// SIMATIC STEP 7 (V5.x) project newgenpns
// station: Hardware
// station: SIMATIC 300(1)
// station: P_ADR_BUS
// station: P_ADR_BUS
// station: Configuration
// program: S7 Program(1)

SYMBOL_TABLE
"PressDB"	DB 3	DB 3
"FCs"	DB 4	DB 4
"NOMINAL"	DB 71	DB 71
"EtoDBfunc"	DB 97	DB 97
"AtoDBfunc"	DB 98	DB 98
"AlarmState"	DB 99	DB 99
"Alarms"	DB 101	DB 101
"mada"	DB 102	DB 102
"Events"	DB 111	DB 111
"DB_ROTATION"	DB 200	DB 200
"PROCESS_DATA"	DB 300	DB 300
"kagiri"	DB 302	DB 302
"DB_PUMPOFF"	DB 303	DB 303
"MM430_NS1"	DB 500	DB 500
"Scale"	FC 3	FC 3
"FaultCheck"	FC 5	FC 5
"DT to DATE"	FC 6	FC 6	// DT to DATE
"DT to DAY"	FC 7	FC 7	// DT to DAY
"DT to TOD"	FC 8	FC 8	// DT to TOD
"GE_DT"	FC 12	FC 12	// Greater or Equal DT
"EventsCheck"	FC 55	FC 55
"DATE and TOD to DT"	FC 62	FC 62	// Date and TOD to DT
"rawConvert"	FC 100	FC 100
"aisConvert"	FC 102	FC 102
"maCalibration"	FC 103	FC 103
"FAULT_CHECK"	FC 105	FC 105
"AlarmToDB"	FC 106	FC 106
"Copyd"	FC 107	FC 107
"ToPanel"	FC 108	FC 108
"EventToDB"	FC 116	FC 116
"Copyb"	FC 117	FC 117
"EToPanel"	FC 118	FC 118
"date&time"	FC 121	FC 121
"ROTATION"	FC 200	FC 200
"PNS_CORE"	FC 300	FC 300
"PUMPS_TOGGLE"	FC 301	FC 301
"FICTION_PRIORITY"	FC 302	FC 302
"MICROMASTER_4XX"	FC 500	FC 500
"Fire"	I 1.0	BOOL
"Security"	I 1.1	BOOL
"Overflow"	I 1.2	BOOL
"Phase"	I 1.3	BOOL
"Input1AVR"	I 2.0	BOOL
"Input2AVR"	I 2.1	BOOL
"Mushroom"	I 2.2	BOOL
"Dryhot"	I 2.3	BOOL
"DI_p1_confirm"	I 3.0	BOOL
"DI_p2_confirm"	I 3.1	BOOL
"DI_p3_confirm"	I 3.2	BOOL
"DI_p4_confirm"	I 3.3	BOOL
"DI_p5_confirm"	I 4.0	BOOL
"DI_p6_confirm"	I 4.1	BOOL
"DI_p1_auto"	I 4.2	BOOL
"DI_p2_auto"	I 4.3	BOOL
"DI_p3_auto"	I 10.0	BOOL
"DI_p4_auto"	I 10.1	BOOL
"pmp1turnOn"	M 13.0	BOOL
"pmp3turnOn"	M 13.1	BOOL
"pmp2turnOn"	M 13.2	BOOL
"RESERVE_BIT"	M 13.3	BOOL
"pmp4turnOn"	M 13.4	BOOL
"SFM0"	M 15.0	BOOL
"SFM1"	M 15.1	BOOL
"SFM2"	M 15.2	BOOL
"SFM3"	M 15.3	BOOL
"EM1"	M 50.0	BOOL
"EM2"	M 50.1	BOOL
"EM3"	M 50.2	BOOL
"EM4"	M 50.3	BOOL
"EM5"	M 50.4	BOOL
"EM6"	M 50.5	BOOL
"EM7"	M 50.6	BOOL
"EM8"	M 50.7	BOOL
"EM9"	M 51.0	BOOL
"EM10"	M 51.1	BOOL
"EM11"	M 51.2	BOOL
"EM12"	M 51.3	BOOL
"starterFPbegin"	M 60.0	BOOL
"starterFPend"	M 60.1	BOOL
"IN_p1_start"	M 70.0	BOOL
"IN_p2_start"	M 70.1	BOOL
"IN_p3_start"	M 70.2	BOOL
"miAuto1"	M 70.3	BOOL
"miAuto2"	M 70.4	BOOL
"miAuto3"	M 70.5	BOOL
"miAuto4"	M 70.6	BOOL
"fcM11"	M 70.7	BOOL
"fcM12"	M 71.0	BOOL
"fcM13"	M 71.1	BOOL
"fcM14"	M 71.2	BOOL
"fcM15"	M 71.3	BOOL
"fcM16"	M 71.4	BOOL
"fcM17"	M 71.5	BOOL
"guuzenFP1"	M 71.6	BOOL
"guuzenFP2"	M 71.7	BOOL
"guuzenFP3"	M 72.0	BOOL
"guuzenFP4"	M 72.1	BOOL
"fcM18"	M 72.2	BOOL
"fcM19"	M 72.3	BOOL
"fcM20"	M 72.4	BOOL
"fcM21"	M 72.5	BOOL
"fcM22"	M 72.6	BOOL
"fcM1"	M 72.7	BOOL
"fcM2"	M 73.0	BOOL
"fcM3"	M 73.1	BOOL
"fcM4"	M 73.2	BOOL
"fcM5"	M 73.3	BOOL
"fcM6"	M 73.4	BOOL
"fcM7"	M 73.5	BOOL
"fcM8"	M 73.6	BOOL
"fcM9"	M 73.7	BOOL
"fcM10"	M 74.0	BOOL
"rotFPbegin"	M 80.0	BOOL
"rotSwiMode"	M 122.0	BOOL
"timeHasCome"	M 122.1	BOOL
"rotation200"	M 122.2	BOOL
"pInput"	PIW 368	WORD
"pOutput"	PIW 370	WORD
"DO_alarm"	Q 4.0	BOOL
"DO_dry"	Q 4.1	BOOL
"DO_p1_turnOn"	Q 6.0	BOOL
"DO_p2_turnOn"	Q 6.1	BOOL
"DO_p3_turnOn"	Q 7.0	BOOL
"DO_p4_turnOn"	Q 7.1	BOOL
"SET_CLK"	SFC 0	SFC 0	// Set System Clock
"READ_CLK"	SFC 1	SFC 1	// Read System Clock
"DPRD_DAT"	SFC 14	SFC 14	// Read Consistent Data of a Standard DP Slave
"DPWR_DAT"	SFC 15	SFC 15	// Write Consistent Data to a Standard DP Slave
"main_started"	T 1	TIMER
"reserve_started"	T 2	TIMER
"lowPressTimer"	T 3	TIMER
"delayStartMain"	T 4	TIMER
"delayStartRes"	T 5	TIMER
"delayStartSRes"	T 6	TIMER
"reserve_stopped"	T 7	TIMER
"second_res_stopped"	T 8	TIMER
"highPressTimer"	T 9	TIMER
"silentRot"	T 10	TIMER
"fcTimer1"	T 13	TIMER
"fcTimer2"	T 14	TIMER
"fcTimer3"	T 15	TIMER
"fcTimer4"	T 16	TIMER
"p2_guuzenTimer"	T 17	TIMER
"p3_guuzenTimer"	T 18	TIMER
"fcTimer9"	T 19	TIMER
"fcTimer10"	T 20	TIMER
"fcTimer5"	T 37	TIMER
"fcTimer6"	T 38	TIMER
"fcTimer7"	T 39	TIMER
"fcTimer8"	T 40	TIMER
"mainFC1_20Hz"	T 41	TIMER
"mainFC2_20Hz"	T 42	TIMER
"mainFC3_20Hz"	T 43	TIMER
"offT0"	T 44	TIMER
"offT1"	T 45	TIMER
"offT2"	T 46	TIMER
"SFoff0"	T 47	TIMER
"SFoff1"	T 48	TIMER
"SFoff2"	T 49	TIMER
"sReserve_started"	T 50	TIMER
"third_res_stopped"	T 51	TIMER
"offT3"	T 52	TIMER
"SFoff3"	T 53	TIMER
END_SYMBOL_TABLE

FUNCTION "Scale" : VOID	// FC 3
TITLE = current to measuring value
VERSION : 1.0
VAR_INPUT
  Current : REAL ;
  STop : REAL ;
  SBottom : REAL ;
END_VAR
VAR_OUTPUT
  Actual_value : REAL ;
END_VAR
VAR_TEMP
  NOENT : REAL ;
END_VAR
BEGIN
NETWORK
TITLE =  Арифметика
// t = SBottom + ((4-Current)*(STop-SBottom))/160
      L     #Current;
      L     4.000000e+00;
      -R;
      T     #NOENT;
      L     #STop;
      L     #SBottom;
      -R;
      L     #NOENT;
      *R;
      L     1.600000e+01;
      /R;
      L     #SBottom;
      +R;
      T     #Actual_value;
END_FUNCTION

FUNCTION "FaultCheck" : VOID	// FC 5
TITLE = Switch to alarm state
VERSION : 0.1
BEGIN
NETWORK
TITLE = check for wirebreak and short of level sensor
      L     DB2.DBD 0;
      L     3.800000e+00;
      <=R;
      L     S5T#1S;
      SD    "fcTimer1";
      A     "fcTimer1";
// =     "AlarmState".BreakIN
// A     "AlarmState".BreakIN
      FP    M 111.0;
      A     M 111.0;
      JCN   brwr;
      CALL  "AlarmToDB" (
           AlarmType                := 1,
           SavLev                   := 0.000000e+00,
           SavCur                   := 0.000000e+00);
brwr: NOP   0;
      L     DB2.DBD 0;
      L     2.100000e+01;
      >R;
      L     S5T#1S;
      SD    "fcTimer2";
      A     "fcTimer2";
//   =     "AlarmState".ShortIN
//  A     "AlarmState".ShortIN
      FP    M 112.0;
      A     M 112.0;
      JCN   shwr;
      CALL  "AlarmToDB" (
           AlarmType                := 2,
           SavLev                   := 0.000000e+00,
           SavCur                   := 0.000000e+00);
shwr: NOP   0;
//  O     "AlarmState".BreakIN
// O     "AlarmState".ShortIN
//S     DB9.DBX   24.2
NETWORK
TITLE = check for wirebreak and short of level sensor
      L     DB2.DBD 4;
      L     3.800000e+00;
      <=R;
      L     S5T#1S;
      SD    "fcTimer9";
      A     "fcTimer9";
      =     "AlarmState".BreakOUT;
      A     "AlarmState".BreakOUT;
      FP    M 202.3;
      A     M 202.3;
      JCN   brwx;
      CALL  "AlarmToDB" (
           AlarmType                := 3,
           SavLev                   := 0.000000e+00,
           SavCur                   := 0.000000e+00);
brwx: NOP   0;
      L     DB2.DBD 4;
      L     2.100000e+01;
      >R;
      L     S5T#1S;
      SD    "fcTimer10";
      A     "fcTimer10";
      =     "AlarmState".ShortOUT;
      A     "AlarmState".ShortOUT;
      FP    M 202.4;
      A     M 202.4;
      JCN   shwx;
      CALL  "AlarmToDB" (
           AlarmType                := 2,
           SavLev                   := 0.000000e+00,
           SavCur                   := 0.000000e+00);
shwx: NOP   0;
//  O     "AlarmState".BreakIN
// O     "AlarmState".ShortIN
//S     DB9.DBX   24.2
NETWORK
TITLE = 12
      AN    "Fire";
//   =     "AlarmState".Fire
      FP    M 116.1;
      A     M 116.1;
      JCN   _000;
      CALL  "AlarmToDB" (
           AlarmType                := 5,
           SavLev                   := 0.000000e+00,
           SavCur                   := 0.000000e+00);
_000: NOP   0;
      AN    "Security";
//  =     "AlarmState".Security
      FP    M 116.2;
      A     M 116.2;
      JCN   _001;
      CALL  "AlarmToDB" (
           AlarmType                := 6,
           SavLev                   := 0.000000e+00,
           SavCur                   := 0.000000e+00);
_001: NOP   0;
      A     "Overflow";
      =     "AlarmState".Flood;
      FP    M 116.3;
      A     M 116.3;
      JCN   _002;
      CALL  "AlarmToDB" (
           AlarmType                := 7,
           SavLev                   := 0.000000e+00,
           SavCur                   := 0.000000e+00);
_002: NOP   0;
      AN    "Phase";
      =     "AlarmState".Phase;
      FP    M 116.4;
      A     M 116.4;
      JCN   _008;
      CALL  "AlarmToDB" (
           AlarmType                := 8,
           SavLev                   := 0.000000e+00,
           SavCur                   := 0.000000e+00);
_008: NOP   0;
NETWORK
TITLE =
//12.07.17 Сухой ход не авария
      A     "Dryhot";
      O;
      A(;
      L     "PressDB".actualPressIN;
      L     "kagiri".shitaKagiriNyuu;
      <=R;
      );
      L     "kagiri".suhoyTime;
      SD    "fcTimer3";
      A     "fcTimer3";
// =     "AlarmState".Dryhod
      =     "DO_dry";
//A     "AlarmState".Dryhod
      A     "DO_dry";
      FP    M 202.5;
      A     M 202.5;
      JCN   dryh;
      CALL  "AlarmToDB" (
           AlarmType                := 12,
           SavLev                   := 0.000000e+00,
           SavCur                   := 0.000000e+00);
dryh: NOP   0;
NETWORK
TITLE = Mushroom
      A     "Mushroom";
      =     "AlarmState".Mushroom;
      FP    M 201.0;
      A     M 201.0;
      JCN   _003;
      CALL  "AlarmToDB" (
           AlarmType                := 11,
           SavLev                   := 0.000000e+00,
           SavCur                   := 0.000000e+00);
_003: NOP   0;
NETWORK
TITLE = saigo
      A     "AtoDBfunc".Allow;
      JCN   allw;
      CALL  "ToPanel";
allw: NOP   0;
      A     I 0.0;
      =     "AtoDBfunc".Allow;
NETWORK
TITLE = sovcim
      L     DB99.DBD 0;
      L     0;
      <>D;
      =     "PROCESS_DATA".Alarma;
      A     "PROCESS_DATA".Alarma;
      =     "DO_alarm";
NETWORK
TITLE = Pmp1off
      A     "DO_p1_turnOn";
      AN    "DI_p1_confirm";
      L     "DB_PUMPOFF".Delay;
      SD    "offT0";
      A     "offT0";
      S     "DB_PUMPOFF".Pmp1off;
NETWORK
TITLE = Pmp2off
      A     "DO_p2_turnOn";
      AN    "DI_p2_confirm";
      L     "DB_PUMPOFF".Delay;
      SD    "offT1";
      A     "offT1";
      S     "DB_PUMPOFF".Pmp2off;
NETWORK
TITLE = Pmp3off
      A     "DO_p3_turnOn";
      AN    "DI_p3_confirm";
      L     "DB_PUMPOFF".Delay;
      SD    "offT2";
      A     "offT2";
      S     "DB_PUMPOFF".Pmp3off;
NETWORK
TITLE = Pmp4off
      A     "DO_p4_turnOn";
      AN    "DI_p4_confirm";
      L     "DB_PUMPOFF".Delay;
      SD    "offT3";
      A     "offT3";
      S     "DB_PUMPOFF".Pmp4off;
NETWORK
TITLE = Pmp1offSF
//      A     "DO_p1_turnOn"
//      AN    "DO_p2_turnOn"
//      AN    "DO_p3_turnOn"
//      AN    "DO_p4_turnOn"
//      A(    
//      L     "PROCESS_DATA".P_setpoint
//      L     "PressDB".actualPressOUT
//      -R    
//      L     "PROCESS_DATA".P_setLowDiff
//      >R    
//      )     
//      L     "DB_PUMPOFF".sf_delay
//      SD    "SFoff0"
//      A     "SFoff0"
//
//      S     "DB_PUMPOFF".Pmp1off
//
//      FP    "SFM0"
//      A     "SFM0"
//
//
//      JCN   _sf0
//
//      CALL  "AlarmToDB"
//       AlarmType:=9
//       SavLev   :="FCs".fc1_currFreq
//       SavCur   :="FCs".fc1_currCurr
//
//
//_sf0: NOP   0
//
//
NETWORK
TITLE = Pmp2offSF
//      A     "DO_p2_turnOn"
//      AN    "DO_p1_turnOn"
//      AN    "DO_p3_turnOn"
//      AN    "DO_p4_turnOn"
//      A(    
//      L     "PROCESS_DATA".P_setpoint
//      L     "PressDB".actualPressOUT
//      -R    
//      L     "PROCESS_DATA".P_setLowDiff
//      >R    
//      )     
//      L     "DB_PUMPOFF".sf_delay
//      SD    "SFoff1"
//      A     "SFoff1"
//
//      S     "DB_PUMPOFF".Pmp2off
//
//      FP    "SFM1"
//      A     "SFM1"
//
//
//      JCN   _sf1
//
//      CALL  "AlarmToDB"
//       AlarmType:=10
//       SavLev   :="FCs".fc2_currFreq
//       SavCur   :="FCs".fc2_currCurr
//
//
//_sf1: NOP   0
//
//
NETWORK
TITLE = Pmp3offSF
//      A     "DO_p3_turnOn"
//      AN    "DO_p1_turnOn"
//      AN    "DO_p2_turnOn"
//      AN    "DO_p4_turnOn"
//      A(    
//      L     "PROCESS_DATA".P_setpoint
//      L     "PressDB".actualPressOUT
//      -R    
//      L     "PROCESS_DATA".P_setLowDiff
//      >R    
//      )     
//      L     "DB_PUMPOFF".sf_delay
//      SD    "SFoff2"
//      A     "SFoff2"
//
//      S     "DB_PUMPOFF".Pmp3off
//
//      FP    "SFM2"
//      A     "SFM2"
//
//
//      JCN   _sf2
//
//      CALL  "AlarmToDB"
//       AlarmType:=13
//       SavLev   :="FCs".fc3_currFreq
//       SavCur   :="FCs".fc3_currCurr
//
//
//_sf2: NOP   0
//
//
NETWORK
TITLE = Pmp4offSF
//      A     "DO_p4_turnOn"
//      AN    "DO_p1_turnOn"
//      AN    "DO_p2_turnOn"
//      AN    "DO_p3_turnOn"
//      A(    
//      L     "PROCESS_DATA".P_setpoint
//      L     "PressDB".actualPressOUT
//      -R    
//      L     "PROCESS_DATA".P_setLowDiff
//      >R    
//      )     
//      L     "DB_PUMPOFF".sf_delay
//      SD    "SFoff3"
//      A     "SFoff3"
//
//      S     "DB_PUMPOFF".Pmp4off
//
//      FP    "SFM3"
//      A     "SFM3"
//
//
//      JCN   _sf3
//
//      CALL  "AlarmToDB"
//       AlarmType:=16
//       SavLev   :="FCs".fc1_currFreq
//       SavCur   :="FCs".fc1_currCurr
//
//
//_sf3: NOP   0
//
//
NETWORK
TITLE =
      A     "DB_PUMPOFF".Pmp1off;
      A     "DB_PUMPOFF".Pmp2off;
      A     "DB_PUMPOFF".Pmp3off;
      A     "DB_PUMPOFF".Pmp4off;
      R     "DB_PUMPOFF".Pmp1off;
      R     "DB_PUMPOFF".Pmp2off;
      R     "DB_PUMPOFF".Pmp3off;
      R     "DB_PUMPOFF".Pmp4off;
END_FUNCTION

// FC 6: know-how protected block, not included

// FC 7: know-how protected block, not included

// FC 8: know-how protected block, not included

// FC 12: know-how protected block, not included

FUNCTION "EventsCheck" : VOID	// FC 55
VERSION : 0.1
BEGIN
NETWORK
TITLE =
      A     "DI_p1_confirm";
      FP    "EM1";
      A     "EM1";
      JCN   eve1;
      CALL  "EventToDB" (
           EventType                := 1);
eve1: NOP   0;
      A     "DI_p2_confirm";
      FP    "EM2";
      A     "EM2";
      JCN   eve2;
      CALL  "EventToDB" (
           EventType                := 2);
eve2: NOP   0;
      A     "DI_p3_confirm";
      FP    "EM3";
      A     "EM3";
      JCN   eve3;
      CALL  "EventToDB" (
           EventType                := 3);
eve3: NOP   0;
      AN    "DI_p1_confirm";
      FP    "EM4";
      A     "EM4";
      JCN   eve4;
      CALL  "EventToDB" (
           EventType                := 4);
eve4: NOP   0;
      AN    "DI_p2_confirm";
      FP    "EM5";
      A     "EM5";
      JCN   eve5;
      CALL  "EventToDB" (
           EventType                := 5);
eve5: NOP   0;
      AN    "DI_p3_confirm";
      FP    "EM6";
      A     "EM6";
      JCN   eve6;
      CALL  "EventToDB" (
           EventType                := 6);
eve6: NOP   0;
NETWORK
TITLE =
      A     "DI_p4_confirm";
      FP    "EM11";
      A     "EM11";
      JCN   eve7;
      CALL  "EventToDB" (
           EventType                := 7);
eve7: NOP   0;
      AN    "DI_p4_confirm";
      FP    "EM12";
      A     "EM12";
      JCN   eve8;
      CALL  "EventToDB" (
           EventType                := 8);
eve8: NOP   0;
NETWORK
TITLE = saigo
      A     "EtoDBfunc".Allow;
      JCN   allw;
      CALL  "EToPanel";
allw: NOP   0;
      A     I 0.0;
      =     "EtoDBfunc".Allow;
END_FUNCTION

// FC 62: know-how protected block, not included

// FC 67: know-how protected block, not included

// FC 70: know-how protected block, not included

FUNCTION "rawConvert" : VOID	// FC 100
TITLE = Преобразование значений каналов
VERSION : 1.0
VAR_INPUT
  Raw : WORD ;	//Считанное аналоговое значение
END_VAR
VAR_OUTPUT
  Current : REAL ;	//Ток в mA
END_VAR
VAR_TEMP
  TDoubleInt : DINT ;
  TInt : INT ;
END_VAR
BEGIN
NETWORK
TITLE =  Преобразование значения в mA
      L     #Raw;
      T     #TInt;
//Только двойные целые могут быть преобразованы в формат REAL
      L     #TInt;
      ITD;
      T     #TDoubleInt;
      L     #TDoubleInt;	//       16-ричное значение
      DTR;	// Ток = --------------------
      T     #Current;	//			    1728
      L     1.728000e+03;	//	!			/
      /R;	//	!		   /
      T     #Current;	//	!		  /
//	+========/===========+===
//			4			20
      L     4.000000e+00;	//Настройка Offset
      +R;
      T     #Current;
END_FUNCTION

FUNCTION "aisConvert" : VOID	// FC 102
TITLE = AIs values convert
VERSION : 1.0
BEGIN
NETWORK
TITLE =  read values from phys channels; convert to mA
      L     "pInput";
      T     DB1.DBW 0;
      L     "pOutput";
      T     DB1.DBW 2;
      CALL  "rawConvert" (
           Raw                      := DB1.DBW 0,
           Current                  := DB2.DBD 0);
      CALL  "rawConvert" (
           Raw                      := DB1.DBW 2,
           Current                  := DB2.DBD 4);
END_FUNCTION

FUNCTION "maCalibration" : VOID	// FC 103
TITLE = current to measuring value
VERSION : 1.0
VAR_INPUT
  Current : REAL ;
  STop : REAL ;
  SBottom : REAL ;
END_VAR
VAR_OUTPUT
  Actual_value : REAL ;
END_VAR
VAR_TEMP
  NOENT : REAL ;
END_VAR
BEGIN
NETWORK
TITLE =  Арифметика
// t = SBottom + ((4-Current)*(STop-SBottom))/160
      L     #Current;
      L     4.000000e+00;
      -R;
      T     #NOENT;
      L     #STop;
      L     #SBottom;
      -R;
      L     #NOENT;
      *R;
      L     1.600000e+01;
      /R;
      L     #SBottom;
      +R;
      T     #Actual_value;
END_FUNCTION

FUNCTION "AlarmToDB" : VOID	// FC 106
VERSION : 0.1
VAR_INPUT
  AlarmType : INT ;
  SavLev : REAL ;
  SavCur : REAL ;
END_VAR
VAR_TEMP
  RTD : DATE_AND_TIME ;
  RT : TIME_OF_DAY ;
  RD : DATE ;
  Num : INT ;
END_VAR
BEGIN
NETWORK
TITLE =
      L     "AtoDBfunc".CurPos;
      L     100;
      ==I;
      JCN   enda;
      L     0;
      T     "AtoDBfunc".CurPos;
enda: NOP   0;
      L     "AtoDBfunc".CurPos;
      INC   1;
      T     "AtoDBfunc".CurPos;
      T     "AtoDBfunc".PanPos;
      T     #Num;
      CALL  "READ_CLK" (
           RET_VAL                  := MW 1,
           CDT                      := #RTD);
      CALL  "DT to DATE" (
           $1                       := #RTD,
           $2                       := #RD);
      CALL  "DT to TOD" (
           $1                       := #RTD,
           $2                       := #RT);
      L     "AtoDBfunc".CurPos;
      L     144;
      *I;
      LAR1;
      OPN   "Alarms";
      L     #Num;
      T     DBW [AR1,P#0.0];
      L     #RD;
      T     DBW [AR1,P#2.0];
      L     #RT;
      T     DBD [AR1,P#4.0];
      L     #AlarmType;
      T     DBW [AR1,P#8.0];
      L     #SavLev;
      T     DBD [AR1,P#10.0];
      L     #SavCur;
      T     DBD [AR1,P#14.0];
      L     "AtoDBfunc".CurPos;
      LAR1;
      OPN   "mada";
      S     DBX [AR1,P#0.0];
      S     "AtoDBfunc".Allow;
END_FUNCTION

FUNCTION "Copyd" : VOID	// FC 107
VERSION : 0.1
VAR_INPUT
  Pos : INT ;
END_VAR
VAR_OUTPUT
  Num : INT ;
  Dat : DATE ;
  Tim : TIME ;
  Typ : INT ;
  Lev : REAL ;
  Cur : REAL ;
END_VAR
BEGIN
NETWORK
TITLE =
      L     #Pos;
      L     144;
      *I;
      LAR1;
      OPN   "Alarms";
      L     DBW [AR1,P#0.0];
      T     #Num;
      L     DBW [AR1,P#2.0];
      T     #Dat;
      L     DBD [AR1,P#4.0];
      T     #Tim;
      L     DBW [AR1,P#8.0];
      T     #Typ;
      L     DBD [AR1,P#10.0];
      T     #Lev;
      L     DBD [AR1,P#14.0];
      T     #Cur;
END_FUNCTION

FUNCTION "ToPanel" : VOID	// FC 108
VERSION : 0.1
BEGIN
NETWORK
TITLE =
//    A     "AtoDBfunc".Qwit
//      JCN   qwi5
//      R     T     37
//      FR    T     37
//      R     T     38
//      FR    T     38
//
//qwi5: NOP   0
//
//
      L     "AtoDBfunc".PanPos;
      L     0;
      <=I;
      JCN   qwer;
      L     100;
      T     "AtoDBfunc".PanPos;
qwer: NOP   0;
      L     "AtoDBfunc".PanPos;
      L     101;
      >=I;
      JCN   qwex;
      L     1;
      T     "AtoDBfunc".PanPos;
qwex: NOP   0;
      CALL  "Copyd" (
           Pos                      := "AtoDBfunc".PanPos,
           Num                      := DB100.DBW 0,
           Dat                      := DB100.DBW 2,
           Tim                      := DB100.DBD 4,
           Typ                      := DB100.DBW 8,
           Lev                      := DB100.DBD 10,
           Cur                      := DB100.DBD 14);
      A     "AtoDBfunc".Qwit;
      JCN   qwit;
      L     "AtoDBfunc".PanPos;
      LAR1;
      OPN   "mada";
      R     DBX [AR1,P#0.0];
qwit: NOP   0;
      L     "AtoDBfunc".PanPos;
      LAR1;
      OPN   "mada";
      A     DBX [AR1,P#0.0];
      =     DB100.DBX 72.0;
      L     "AtoDBfunc".PanPos;
      T     LW 1;
      L     1;
      ==I;
      JCN   srts;
      L     101;
      T     LW 1;
srts: L     LW 1;
      DEC   1;
      T     LW 1;
      CALL  "Copyd" (
           Pos                      := LW 1,
           Num                      := DB100.DBW 18,
           Dat                      := DB100.DBW 20,
           Tim                      := DB100.DBD 22,
           Typ                      := DB100.DBW 26,
           Lev                      := DB100.DBD 28,
           Cur                      := DB100.DBD 32);
      A     "AtoDBfunc".Qwit;
      JCN   qwi2;
      L     LW 1;
      LAR1;
      OPN   "mada";
      R     DBX [AR1,P#0.0];
qwi2: NOP   0;
      L     LW 1;
      LAR1;
      OPN   "mada";
      A     DBX [AR1,P#0.0];
      =     DB100.DBX 72.1;
      L     LW 1;
      L     1;
      ==I;
      JCN   srtf;
      L     101;
      T     LW 1;
srtf: L     LW 1;
      DEC   1;
      T     LW 1;
      CALL  "Copyd" (
           Pos                      := LW 1,
           Num                      := DB100.DBW 36,
           Dat                      := DB100.DBW 38,
           Tim                      := DB100.DBD 40,
           Typ                      := DB100.DBW 44,
           Lev                      := DB100.DBD 46,
           Cur                      := DB100.DBD 50);
      A     "AtoDBfunc".Qwit;
      JCN   qwi3;
      L     LW 1;
      LAR1;
      OPN   "mada";
      R     DBX [AR1,P#0.0];
qwi3: NOP   0;
      L     LW 1;
      LAR1;
      OPN   "mada";
      A     DBX [AR1,P#0.0];
      =     DB100.DBX 72.2;
      L     LW 1;
      L     1;
      ==I;
      JCN   srtx;
      L     101;
      T     LW 1;
srtx: L     LW 1;
      DEC   1;
      T     LW 1;
      CALL  "Copyd" (
           Pos                      := LW 1,
           Num                      := DB100.DBW 54,
           Dat                      := DB100.DBW 56,
           Tim                      := DB100.DBD 58,
           Typ                      := DB100.DBW 62,
           Lev                      := DB100.DBD 64,
           Cur                      := DB100.DBD 68);
      A     "AtoDBfunc".Qwit;
      JCN   qwi4;
      L     LW 1;
      LAR1;
      OPN   "mada";
      R     DBX [AR1,P#0.0];
qwi4: NOP   0;
      L     LW 1;
      LAR1;
      OPN   "mada";
      A     DBX [AR1,P#0.0];
      =     DB100.DBX 72.3;
      A     I 0.0;
      =     "AtoDBfunc".Qwit;
END_FUNCTION

FUNCTION "EventToDB" : VOID	// FC 116
VERSION : 0.1
VAR_INPUT
  EventType : INT ;
END_VAR
VAR_TEMP
  RTD : DATE_AND_TIME ;
  RT : TIME_OF_DAY ;
  RD : DATE ;
  Num : INT ;
END_VAR
BEGIN
NETWORK
TITLE =
      L     "EtoDBfunc".CurPos;
      L     100;
      ==I;
      JCN   enda;
      L     0;
      T     "EtoDBfunc".CurPos;
enda: NOP   0;
      L     "EtoDBfunc".CurPos;
      INC   1;
      T     "EtoDBfunc".CurPos;
      T     "EtoDBfunc".PanPos;
      T     #Num;
      CALL  "READ_CLK" (
           RET_VAL                  := MW 1,
           CDT                      := #RTD);
      CALL  "DT to DATE" (
           $1                       := #RTD,
           $2                       := #RD);
      CALL  "DT to TOD" (
           $1                       := #RTD,
           $2                       := #RT);
      L     "EtoDBfunc".CurPos;
      L     80;
      *I;
      LAR1;
      OPN   "Events";
      L     #Num;
      T     DBW [AR1,P#0.0];
      L     #RD;
      T     DBW [AR1,P#2.0];
      L     #RT;
      T     DBD [AR1,P#4.0];
      L     #EventType;
      T     DBW [AR1,P#8.0];
      S     "EtoDBfunc".Allow;
END_FUNCTION

FUNCTION "Copyb" : VOID	// FC 117
VERSION : 0.1
VAR_INPUT
  Pos : INT ;
END_VAR
VAR_OUTPUT
  Num : INT ;
  Dat : DATE ;
  Tim : TIME ;
  Typ : INT ;
END_VAR
BEGIN
NETWORK
TITLE =
      L     #Pos;
      L     80;
      *I;
      LAR1;
      OPN   "Events";
      L     DBW [AR1,P#0.0];
      T     #Num;
      L     DBW [AR1,P#2.0];
      T     #Dat;
      L     DBD [AR1,P#4.0];
      T     #Tim;
      L     DBW [AR1,P#8.0];
      T     #Typ;
END_FUNCTION

FUNCTION "EToPanel" : VOID	// FC 118
VERSION : 0.1
BEGIN
NETWORK
TITLE =
      L     "EtoDBfunc".PanPos;
      L     0;
      <=I;
      JCN   qwer;
      L     100;
      T     "EtoDBfunc".PanPos;
qwer: NOP   0;
      L     "EtoDBfunc".PanPos;
      L     101;
      >=I;
      JCN   qwex;
      L     1;
      T     "EtoDBfunc".PanPos;
qwex: NOP   0;
      CALL  "Copyb" (
           Pos                      := "EtoDBfunc".PanPos,
           Num                      := DB112.DBW 0,
           Dat                      := DB112.DBW 2,
           Tim                      := DB112.DBD 4,
           Typ                      := DB112.DBW 8);
      L     "EtoDBfunc".PanPos;
      T     LW 11;
      L     1;
      ==I;
      JCN   srts;
      L     101;
      T     LW 11;
srts: L     LW 11;
      DEC   1;
      T     LW 11;
      CALL  "Copyb" (
           Pos                      := LW 11,
           Num                      := DB112.DBW 10,
           Dat                      := DB112.DBW 12,
           Tim                      := DB112.DBD 14,
           Typ                      := DB112.DBW 18);
      L     LW 11;
      L     1;
      ==I;
      JCN   srtf;
      L     101;
      T     LW 11;
srtf: L     LW 11;
      DEC   1;
      T     LW 11;
      CALL  "Copyb" (
           Pos                      := LW 11,
           Num                      := DB112.DBW 20,
           Dat                      := DB112.DBW 22,
           Tim                      := DB112.DBD 24,
           Typ                      := DB112.DBW 28);
      L     LW 11;
      L     1;
      ==I;
      JCN   srtx;
      L     101;
      T     LW 11;
srtx: L     LW 11;
      DEC   1;
      T     LW 11;
      CALL  "Copyb" (
           Pos                      := LW 11,
           Num                      := DB112.DBW 30,
           Dat                      := DB112.DBW 32,
           Tim                      := DB112.DBD 34,
           Typ                      := DB112.DBW 38);
END_FUNCTION

FUNCTION "date&time" : VOID	// FC 121
VERSION : 0.1
VAR_TEMP
  RealDT : DATE_AND_TIME ;
  DATETIME : DATE_AND_TIME ;
END_VAR
BEGIN
NETWORK
TITLE =
// A     DB13.DBX    0.6
//      JCN   end
//
//      CALL  "DATE and TOD to DT"
//       IN1    :=DB13.DBW12              //Соединяем дату и время
//       IN2    :=DB13.DBD8
//       RET_VAL:=#DATETIME
//
//      CALL  "SET_CLK"
//       PDT    :=#DATETIME
//       RET_VAL:=MW1
//
//      R     DB13.DBX    0.6             //Reset
//
//end:  NOP   0
//
      CALL  "READ_CLK" (
           RET_VAL                  := MW 1,
           CDT                      := #RealDT);	//Текущие время и дата
      CALL  FC 70 (
           $1                       := #RealDT,
           $2                       := DB13.DBD 2);
      CALL  FC 67 (
           $1                       := #RealDT,
           $2                       := DB13.DBW 6);
      A     DB13.DBX 0.0;
      JCN   end;
      CALL  "DATE and TOD to DT" (
           $1                       := DB13.DBW 12,
           $2                       := DB13.DBD 8,
           $3                       := #DATETIME);	//Соединяем дату и время
      CALL  "SET_CLK" (
           PDT                      := #DATETIME,
           RET_VAL                  := MW 1);
      R     DB13.DBX 0.0;	//Reset
end:  NOP   0;
END_FUNCTION

FUNCTION "ROTATION" : VOID	// FC 200
//27.09.16 -- добавлен 4й НА
//
AUTHOR : rooman
VERSION : 0.1
VAR_INPUT
  p1_DI_auto : BOOL ;
  p2_DI_auto : BOOL ;
  p3_DI_auto : BOOL ;
  p4_DI_auto : BOOL ;
END_VAR
VAR_OUTPUT
  p1_iAuto : BOOL ;
  p2_iAuto : BOOL ;
  p3_iAuto : BOOL ;
  p4_iAuto : BOOL ;
END_VAR
VAR_TEMP
  realDT : DATE_AND_TIME ;
  orderDT : DATE_AND_TIME ;
  realD : DATE ;
  today : INT ;	//rotSwiMode : BOOL;
//timeHasCome : BOOL;
//rotation : BOOL;
END_VAR
BEGIN
NETWORK
TITLE =
//ждем наступления момента Х
      CALL  "READ_CLK" (
           RET_VAL                  := MW 0,
           CDT                      := #realDT);
      CALL  "DT to DATE" (
           $1                       := #realDT,
           $2                       := #realD);
      CALL  "DATE and TOD to DT" (
           $1                       := #realD,
           $2                       := "DB_ROTATION".swiTime,
           $3                       := #orderDT);
      CALL  "GE_DT" (
           $1                       := #realDT,
           $2                       := #orderDT,
           $3                       := "timeHasCome");
      CALL  "DT to DAY" (
           $1                       := #realDT,
           $2                       := #today);
NETWORK
TITLE =
//включаем режим переключения комбинации
      L     #today;
      L     1;
      -I;
      LAR1;
      OPN   "DB_ROTATION";
      A     DBX [AR1,P#0.0];
      A     "timeHasCome";
      FP    "rotFPbegin";
      S     "rotSwiMode";
      S     "rotation200";
NETWORK
TITLE =
//если режим переключения включен, гасим НА
      A     "rotSwiMode";
      JCN   _000;
      CLR;
      =     #p1_iAuto;
      =     #p2_iAuto;
      =     #p3_iAuto;
      =     #p4_iAuto;
_000: NOP   0;
NETWORK
TITLE =
//в противном случае используем команды с галетников
      AN    "rotSwiMode";
      JCN   _001;
      A     #p1_DI_auto;
      =     #p1_iAuto;
      A     #p2_DI_auto;
      =     #p2_iAuto;
      A     #p3_DI_auto;
      =     #p3_iAuto;
      A     #p4_DI_auto;
      =     #p4_iAuto;
_001: NOP   0;
NETWORK
TITLE =
//запускаем таймер
      A     "rotSwiMode";
      L     "DB_ROTATION".silentHill;
      SD    "silentRot";
NETWORK
TITLE =
//ротация лол
      A(;
      A     "rotation200";
      A     "DB_ROTATION".prioScheme_1;
      );
      JCN   _005;
      R     "rotation200";
      R     "DB_ROTATION".prioScheme_1;
      S     "DB_ROTATION".prioScheme_2;
_005: NOP   0;
NETWORK
TITLE =
//ротация
      A(;
      A     "rotation200";
      A     "DB_ROTATION".prioScheme_2;
      );
      JCN   _006;
      R     "rotation200";
      R     "DB_ROTATION".prioScheme_2;
      S     "DB_ROTATION".prioScheme_3;
_006: NOP   0;
NETWORK
TITLE =
//ротация
      A(;
      A     "rotation200";
      A     "DB_ROTATION".prioScheme_3;
      );
      JCN   _007;
      R     "rotation200";
      R     "DB_ROTATION".prioScheme_3;
      S     "DB_ROTATION".prioScheme_4;
_007: NOP   0;
NETWORK
TITLE =
//ротация
      A(;
      A     "rotation200";
      A     "DB_ROTATION".prioScheme_4;
      );
      JCN   _071;
      R     "rotation200";
      R     "DB_ROTATION".prioScheme_4;
      S     "DB_ROTATION".prioScheme_1;
_071: NOP   0;
NETWORK
TITLE =
//используем схему 1
      A(;
      AN    "DI_p1_confirm";
      AN    "DI_p2_confirm";
      AN    "DI_p3_confirm";
      AN    "DI_p4_confirm";
      A     "DB_ROTATION".prioScheme_1;
      );
      JCN   _002;
      L     1;
      T     "PROCESS_DATA".p1_priority;
      L     2;
      T     "PROCESS_DATA".p2_priority;
      L     3;
      T     "PROCESS_DATA".p3_priority;
//L 4;
//T #PROCESS_DATA.p4_priority; 28.12.2016
      L     4;
      T     "PROCESS_DATA".p4_priority;
_002: NOP   0;
NETWORK
TITLE =
//2
      A(;
      AN    "DI_p1_confirm";
      AN    "DI_p2_confirm";
      AN    "DI_p3_confirm";
      AN    "DI_p4_confirm";
      A     "DB_ROTATION".prioScheme_2;
      );
      JCN   _003;
      L     3;	// 28.12.2016
      T     "PROCESS_DATA".p1_priority;
      L     1;
      T     "PROCESS_DATA".p2_priority;
      L     2;
      T     "PROCESS_DATA".p3_priority;
//L 3;
//T #PROCESS_DATA.p4_priority; 28.12.2016
      L     4;
      T     "PROCESS_DATA".p4_priority;
_003: NOP   0;
NETWORK
TITLE =
//3
      A(;
      AN    "DI_p1_confirm";
      AN    "DI_p2_confirm";
      AN    "DI_p3_confirm";
      AN    "DI_p4_confirm";
      A     "DB_ROTATION".prioScheme_3;
      );
      JCN   _004;
      L     2;	// 28.12.2016
      T     "PROCESS_DATA".p1_priority;
      L     3;	// 28.12.2016
      T     "PROCESS_DATA".p2_priority;
      L     1;
      T     "PROCESS_DATA".p3_priority;
//L 2;
//T #PROCESS_DATA.p4_priority; 28.12.2016
      L     4;
      T     "PROCESS_DATA".p4_priority;
_004: NOP   0;
NETWORK
TITLE =
//4
      A(;
      AN    "DI_p1_confirm";
      AN    "DI_p2_confirm";
      AN    "DI_p3_confirm";
      AN    "DI_p4_confirm";
      A     "DB_ROTATION".prioScheme_4;
      );
      JCN   _040;
      L     2;	// 28.12.2016
      T     "PROCESS_DATA".p1_priority;
      L     1;	// 28.12.2016
      T     "PROCESS_DATA".p2_priority;
      L     3;	// 28.12.2016
      T     "PROCESS_DATA".p3_priority;
//L 1;
//T #PROCESS_DATA.p4_priority; 28.12.2016
      L     4;
      T     "PROCESS_DATA".p4_priority;
_040: NOP   0;
NETWORK
TITLE =
//если таймер всё, отключаем режим
      A     "silentRot";
      R     "rotSwiMode";
NETWORK
TITLE =
//разрешение переключения кобинаций
      A(;
      AN    "DI_p1_confirm";
      AN    "DI_p2_confirm";
      AN    "DI_p3_confirm";
      AN    "DI_p4_confirm";
      );
      =     "DB_ROTATION".allow;
NETWORK
TITLE =
//если не выбрана никакая схема, выбираем первую 03.02.16 //27.09.16
      AN    "DB_ROTATION".prioScheme_1;
      AN    "DB_ROTATION".prioScheme_2;
      AN    "DB_ROTATION".prioScheme_3;
      AN    "DB_ROTATION".prioScheme_4;
      S     "DB_ROTATION".prioScheme_1;
END_FUNCTION

FUNCTION "PNS_CORE" : VOID	// FC 300
AUTHOR : rooman
VERSION : 0.1
VAR_INPUT
  p1_iAuto : BOOL ;	//команда на включение насоса в авто-режиме
  p1_confirm : BOOL ;
  p2_iAuto : BOOL ;
  p2_confirm : BOOL ;
  p3_iAuto : BOOL ;
  p3_confirm : BOOL ;
  p4_iAuto : BOOL ;	//26.09.16
  p4_confirm : BOOL ;
  P_current : REAL ;	//fc1_curFreq : REAL;
//fc2_curFreq	: REAL;
//fc3_curFreq : REAL;
  p1_ficPrior : INT ;
  p2_ficPrior : INT ;
  p3_ficPrior : INT ;
  p4_ficPrior : INT ;
END_VAR
VAR_OUTPUT
  p1_oWithFC : BOOL ;
  p2_oWithFC : BOOL ;	//p2_oDirect	: BOOL;
  p3_oWithFC : BOOL ;	//p3_oDirect	: BOOL;
  p4_out : BOOL ;
  fc1_oSetP : REAL ;
  fc2_oSetP : REAL ;
  fc3_oSetP : REAL ;
END_VAR
VAR_TEMP
  mainMustStart : BOOL ;
  resMustStart : BOOL ;
  sResMustStart : BOOL ;
  thResMustStart : BOOL ;	//sResStartMode : BOOL;
//allowDirect	  : BOOL;
//p1_ficPrior		: INT;
//p2_ficPrior		:
END_VAR
BEGIN
NETWORK
TITLE =
//---------------------------включение НА в авто внезапно--------------------
//NETWORK
//TITLE =
////запрет включения второго НА, если третий работает от ПЧ
//	A #p2_iAuto;
//	FP #guuzenFP1;
//	A(;
//		L #PROCESS_DATA.p2_priority;
//		L #PROCESS_DATA.p3_priority;
//		<I;
//		);
//	A #p3_oWithFC;
//	L S5T#15S;
//	SF #p2_guuzenTimer;
//	
//NETWORK
//TITLE =
////запрет включения третьего НА, если второй работает от ПЧ
//
//	A #p3_iAuto;
//	FP #guuzenFP2;
//	A(;
//		L #PROCESS_DATA.p2_priority;
//		L #PROCESS_DATA.p3_priority;
//		>I;
//		);
//	A #p2_oWithFC;
//	L S5T#15S;
//	SF #p3_guuzenTimer;
//	
//NETWORK
//TITLE =
////
//	A #p2_iAuto;
//	FN #guuzenFP3;
//	A(;
//		L #PROCESS_DATA.p2_priority;
//		L #PROCESS_DATA.p3_priority;
//		<I;
//		);
//	AN #p3_oWithFC;
//	L S5T#15S;
//	SF #p3_guuzenTimer;
//
//NETWORK
//TITLE =
////
//
//	A #p3_iAuto;
//	FN #guuzenFP4;
//	A(;
//		L #PROCESS_DATA.p2_priority;
//		L #PROCESS_DATA.p3_priority;
//		>I;
//		);
//	AN #p2_oWithFC;
//	L S5T#15S;
//	SF #p2_guuzenTimer;
//
//--------------------------------END_GUUZEN---------------------------------
//---------------------проверка необходимости включения НАs-----------------
NETWORK
TITLE =
//проверка низкого давления относительно уставки
      A(;
      L     "PROCESS_DATA".P_setpoint;
      L     #P_current;
      -R;
      L     "PROCESS_DATA".P_setLowDiff;
      >R;
      );
      L     "PROCESS_DATA".delayLow;
      SD    "lowPressTimer";
NETWORK
TITLE =
//проверка высокого давления
      A(;
      L     #P_current;
      L     "PROCESS_DATA".P_setpoint;
      -R;
      L     "PROCESS_DATA".P_setUpDiff;
      >R;
      );
      L     "PROCESS_DATA".delayUp;
      SD    "highPressTimer";
//--------------------проверка 20 Гц-------------14.01.2016--------------
NETWORK
TITLE =
//если первый ПЧ некоторое время работает на 20 Гц, то запускаем таймер
//
//A #mainMustStart;
//A #DO_p1_turnOn;
      A     "DI_p1_confirm";
      A(;
      AN    "DI_p2_confirm";
      AN    "DI_p3_confirm";
      );
      A(;
      L     "FCs".fc1_currFreq;
      L     "PROCESS_DATA".lowerHz;
      <R;
      );
      L     "PROCESS_DATA".TwentyHzOffDelay;
      SD    "mainFC1_20Hz";
NETWORK
TITLE =
//если второй насос с ПЧ некоторое время работает на 20 Гц, то запускаем таймер				
//
//A #mainMustStart;
//A #DO_p2_turnOnFC;
      A     "DI_p2_confirm";
      A(;
      AN    "DI_p1_confirm";
      AN    "DI_p3_confirm";
      );
      A(;
      L     "FCs".fc1_currFreq;
      L     "PROCESS_DATA".lowerHz;
      <R;
      );
      L     "PROCESS_DATA".TwentyHzOffDelay;
      SD    "mainFC2_20Hz";
NETWORK
TITLE =
//если третий насос с ПЧ некоторое время работает на 20 Гц, то запускаем таймер
//
//A #mainMustStart;
//A #DO_p3_turnOnFC;
      A     "DI_p3_confirm";
      A(;
      AN    "DI_p1_confirm";
      AN    "DI_p2_confirm";
      );
      A(;
      L     "FCs".fc1_currFreq;
      L     "PROCESS_DATA".lowerHz;
      <R;
      );
      L     "PROCESS_DATA".TwentyHzOffDelay;
      SD    "mainFC3_20Hz";
//---------------------------------------------------------------------
NETWORK
TITLE =
//функция, определяющая необходимость запуска основного и резервных НА
//p1_iAuto	:= p1_iAuto,
      CALL  "PUMPS_TOGGLE" (
           p1_confirm               := #p1_confirm,
           p2_confirm               := #p2_confirm,
           p3_confirm               := #p3_confirm,
           p4_confirm               := #p4_confirm,
           p1_priority              := #p1_ficPrior,
           p2_priority              := #p2_ficPrior,
           p3_priority              := #p3_ficPrior,
           p4_priority              := #p4_ficPrior,
           delayPump                := "PROCESS_DATA".delayPump,
           P_current                := #P_current,
           P_setpoint               := "PROCESS_DATA".P_setpoint,
           mainMustStart            := #mainMustStart,
           resMustStart             := #resMustStart,
           sResMustStart            := #sResMustStart,
           thResMustStart           := #thResMustStart);
//--------------------------------запуск НАs от ПЧ-------------------------------
NETWORK
TITLE =
//запуск первого насоса с ПЧ
      A     #p1_iAuto;
      A(;
      O(;
      L     1;
      L     #p1_ficPrior;
      ==I;
      A     #mainMustStart;
      );
      O(;
      L     2;
      L     #p1_ficPrior;
      ==I;
      A     #resMustStart;
      );
      O(;
      L     3;
      L     #p1_ficPrior;
      ==I;
      A     #sResMustStart;
      );
      O(;
      L     4;
      L     #p1_ficPrior;
      ==I;
      A     #thResMustStart;
      );
      );
      =     #p1_oWithFC;
NETWORK
TITLE =
//запуск второго насоса с ПЧ
      A     #p2_iAuto;
      A(;
      O(;
      L     1;
      L     #p2_ficPrior;
      ==I;
      A     #mainMustStart;
      );
      O(;
      L     2;
      L     #p2_ficPrior;
      ==I;
      A     #resMustStart;
      );
      O(;
      L     3;
      L     #p2_ficPrior;
      ==I;
      A     #sResMustStart;
      );
      O(;
      L     4;
      L     #p2_ficPrior;
      ==I;
      A     #thResMustStart;
      );
      );
//AN #p2_guuzenTimer;
      =     #p2_oWithFC;
NETWORK
TITLE =
//запуск третьего насоса с ПЧ
      A     #p3_iAuto;
      A(;
      O(;
      L     1;
      L     #p3_ficPrior;
      ==I;
      A     #mainMustStart;
      );
      O(;
      L     2;
      L     #p3_ficPrior;
      ==I;
//A #p1_iAuto;
      A     #resMustStart;
      );
      O(;
      L     3;
      L     #p3_ficPrior;
      ==I;
      A     #sResMustStart;
      );
      O(;
      L     4;
      L     #p3_ficPrior;
      ==I;
      A     #thResMustStart;
      );
      );
//AN #p3_guuzenTimer;
      =     #p3_oWithFC;
NETWORK
TITLE =
//запуск четвертого насоса с ПЧ
      A     #p4_iAuto;
      A(;
      O(;
      L     1;
      L     #p4_ficPrior;
      ==I;
      A     #mainMustStart;
      );
      O(;
      L     2;
      L     #p4_ficPrior;
      ==I;
//A #p1_iAuto;
      A     #resMustStart;
      );
      O(;
      L     3;
      L     #p4_ficPrior;
      ==I;
      A     #sResMustStart;
      );
      O(;
      L     4;
      L     #p4_ficPrior;
      ==I;
      A     #thResMustStart;
      );
      );
//AN #p3_guuzenTimer;
      =     #p4_out;
//----------------------процесс запуска НА2,3 от пускателя-----------------------
//NETWORK
//TITLE =
////начало запуска второго резервного
//
//	A #DI_p2_auto;
//	A #DI_p3_auto;
//	A(;
//		O #sResMustStart;
//		O(;
//			AN #p1_iAuto;
//			A #resMustStart;
//		);
//	);
//	//FP #starterFPbegin;
//	S #sResStartMode;
//	
//NETWORK
//TITLE =
////сброс режима включения второго резервного
//	O #p2_oDirect;
//	O #p3_oDirect;
//	//FP #starterFPend;
//		
//	R #sResStartMode;	
//		      
//
//NETWORK
//TITLE =
////расчет фиктивной уставки
//	L #PROCESS_DATA.P_setpoint;
//	A #sResStartMode;
//	JCN _307;
//	
//		L #P_current;
//		L #PROCESS_DATA.P_deltaFic;
//		-R;
//	
//		L 0.000000e+000;
//		<R;			
//		JC _306;
//			TAK;
//		_306: NOP 0;
//
//	_307: NOP 0;
//	T #fc1_oSetP;
//	T #fc2_oSetP;
//	
//NETWORK
//TITLE =
////проверка возможности включения второго резервного ( от пускателя )
//
//	A #sResStartMode;
//	A(;
//		L #fc1_curFreq;
//		L #PROCESS_DATA.alloDirFreq;
//		<=R;
//	);
//	A(;
//		L #fc2_curFreq;
//		L #PROCESS_DATA.alloDirFreq;
//		<=R;
//	);
//	
//	= #allowDirect;
//	
//NETWORK
//TITLE =
////включение НА2 от пускателя
//	A #PROCESS_DATA.allowSecRes;
//	A #p2_iAuto;
//	A(;
//		L 3;
//		L #p2_ficPrior;
//		==I;
//	);
//	A #sResMustStart;
//	A(;
//		O #allowDirect;
//		O #p2_oDirect;
//	);
//	
//	= #p2_oDirect;
//	
//NETWORK
//TITLE =
////включение НА3 от пускателя
//	A #PROCESS_DATA.allowSecRes;
//	A #p3_iAuto;
//	A(;
//		L 3;
//		L #p3_ficPrior;
//		==I;
//		O(;
//			L 2;
//			L #p3_ficPrior;
//			==I;
//			AN #p1_iAuto;
//		);
//	);
//	A(;
//		O #sResMustStart;
//		O(;
//			A #resMustStart;
//			AN #p1_iAuto;
//		);
//	);
//	A(;
//		O #allowDirect;
//		O #p3_oDirect;
//	);
//	
//	= #p3_oDirect;
//	
//END_FUNCTION
//-----------------------------------------------------------------
NETWORK
TITLE =
//уставка
      L     "PROCESS_DATA".P_setpoint;
      T     #fc1_oSetP;
      T     #fc2_oSetP;
      T     #fc3_oSetP;
END_FUNCTION

FUNCTION "PUMPS_TOGGLE" : VOID	// FC 301
AUTHOR : rooman
VERSION : 0.1
VAR_INPUT
  p1_confirm : BOOL ;
  p2_confirm : BOOL ;
  p3_confirm : BOOL ;
  p4_confirm : BOOL ;
  p1_priority : INT ;
  p2_priority : INT ;
  p3_priority : INT ;
  p4_priority : INT ;
  delayPump : S5TIME ;
  P_current : REAL ;	//??
  P_setpoint : REAL ;
END_VAR
VAR_OUTPUT
  mainMustStart : BOOL ;
  resMustStart : BOOL ;
  sResMustStart : BOOL ;
  thResMustStart : BOOL ;
END_VAR
VAR_TEMP
  resConOut : BOOL ;
  sResConOut : BOOL ;
  thResConOut : BOOL ;	//sResStarted : BOOL;
  thResStarted : BOOL ;
  mainStopped : BOOL ;
  mainConfirm : BOOL ;
  resConfirm : BOOL ;
  sResConfirm : BOOL ;
  mainMustStop : BOOL ;
  resMustStop : BOOL ;
  sResMustStop : BOOL ;
  thResMustStop : BOOL ;
END_VAR
BEGIN
NETWORK
TITLE =
//считаем количество НА в стопе 28.12.2016
      L     0;
      T     "PROCESS_DATA".autoCount;
      A     "DI_p1_auto";
      JC    _cn1;
      L     "PROCESS_DATA".autoCount;
      INC   1;
      T     "PROCESS_DATA".autoCount;
_cn1: NOP   0;
      A     "DI_p2_auto";
      JC    _cn2;
      L     "PROCESS_DATA".autoCount;
      INC   1;
      T     "PROCESS_DATA".autoCount;
_cn2: NOP   0;
      A     "DI_p3_auto";
      JC    _cn3;
      L     "PROCESS_DATA".autoCount;
      INC   1;
      T     "PROCESS_DATA".autoCount;
_cn3: NOP   0;
      A     "DI_p4_auto";
      JC    _cn4;
      L     "PROCESS_DATA".autoCount;
      INC   1;
      T     "PROCESS_DATA".autoCount;
_cn4: NOP   0;
NETWORK
TITLE =
//таймер для запуска первого резервного насоса
      O(;
      L     #p1_priority;
      L     1;
      ==I;
      A     #p1_confirm;
      );
      O(;
      L     #p2_priority;
      L     1;
      ==I;
      A     #p2_confirm;
      );
      O(;
      L     #p3_priority;
      L     1;
      ==I;
      A     #p3_confirm;
      );
      O(;
      L     #p4_priority;
      L     1;
      ==I;
      A     #p4_confirm;
      );
      =     #mainConfirm;
      L     #delayPump;
      SD    "main_started";
NETWORK
TITLE =
//таймер для запуска второго резервного насоса	
      O(;
      L     #p1_priority;
      L     2;
      ==I;
      A     #p1_confirm;
      );
      O(;
      L     #p2_priority;
      L     2;
      ==I;
      A     #p2_confirm;
      );
      O(;
      L     #p3_priority;
      L     2;
      ==I;
      A     #p3_confirm;
      );
      O(;
      L     #p4_priority;
      L     2;
      ==I;
      A     #p4_confirm;
      );
      =     #resConfirm;
      L     #delayPump;
      SD    "reserve_started";
NETWORK
TITLE =
//таймер для запуска третьего резервного насоса	
      O(;
      L     #p1_priority;
      L     3;
      ==I;
      A     #p1_confirm;
      );
      O(;
      L     #p2_priority;
      L     3;
      ==I;
      A     #p2_confirm;
      );
      O(;
      L     #p3_priority;
      L     3;
      ==I;
      A     #p3_confirm;
      );
      O(;
      L     #p4_priority;
      L     3;
      ==I;
      A     #p4_confirm;
      );
      =     #sResConfirm;
      L     #delayPump;
      SD    "sReserve_started";
NETWORK
TITLE =
//третий резервный запущен
      O(;
      L     #p1_priority;
      L     4;
      ==I;
      A     #p1_confirm;
      );
      O(;
      L     #p2_priority;
      L     4;
      ==I;
      A     #p2_confirm;
      );
      O(;
      L     #p3_priority;
      L     4;
      ==I;
      A     #p3_confirm;
      );
      O(;
      L     #p4_priority;
      L     4;
      ==I;
      A     #p4_confirm;
      );
      =     #thResStarted;
NETWORK
TITLE =
//таймер после останова третьего резервного
      O(;
      L     #p1_priority;
      L     4;
      ==I;
      AN    #p1_confirm;
      );
      O(;
      L     #p2_priority;
      L     4;
      ==I;
      AN    #p2_confirm;
      );
      O(;
      L     #p3_priority;
      L     4;
      ==I;
      AN    #p3_confirm;
      );
      O(;
      L     #p4_priority;
      L     4;
      ==I;
      AN    #p4_confirm;
      );
      =     #thResConOut;
      L     #delayPump;
      SD    "third_res_stopped";
NETWORK
TITLE =
//таймер после останова второго резервного
      O(;
      L     #p1_priority;
      L     3;
      ==I;
      AN    #p1_confirm;
      );
      O(;
      L     #p2_priority;
      L     3;
      ==I;
      AN    #p2_confirm;
      );
      O(;
      L     #p3_priority;
      L     3;
      ==I;
      AN    #p3_confirm;
      );
      O(;
      L     #p4_priority;
      L     3;
      ==I;
      AN    #p4_confirm;
      );
// не понимаю, но оставлю на всякий случай
//	O(;
//		L #p3_priority;
//		L 2;
//		==I;
//		AN #p1_iAuto;
//	);
      =     #sResConOut;
      L     #delayPump;
      SD    "second_res_stopped";
NETWORK
TITLE =
//таймер после останова резервного
      O(;
      L     #p1_priority;
      L     2;
      ==I;
      AN    #p1_confirm;
      );
      O(;
      L     #p2_priority;
      L     2;
      ==I;
      AN    #p2_confirm;
      );
      O(;
      L     #p3_priority;
      L     2;
      ==I;
      AN    #p3_confirm;
      );
      O(;
      L     #p4_priority;
      L     2;
      ==I;
      AN    #p4_confirm;
      );
      =     #resConOut;
      L     #delayPump;
      SD    "reserve_stopped";
NETWORK
TITLE =
//основной остановлен
      O(;
      L     #p1_priority;
      L     1;
      ==I;
      AN    #p1_confirm;
      );
      O(;
      L     #p2_priority;
      L     1;
      ==I;
      AN    #p2_confirm;
      );
      O(;
      L     #p3_priority;
      L     1;
      ==I;
      AN    #p3_confirm;
      );
      O(;
      L     #p4_priority;
      L     1;
      ==I;
      AN    #p4_confirm;
      );
      =     #mainStopped;
NETWORK
TITLE =
//запрос останова основного НА
      O(;
      A     "main_started";
      A(;
      O     "reserve_stopped";
      O(;
      L     "PROCESS_DATA".autoCount;
      L     3;
      ==I;
      );
      );
      A     "highPressTimer";
      );
      O(;
      A     #mainStopped;
      AN    #mainMustStart;
      );
      O(;
      O     "mainFC1_20Hz";
      O     "mainFC2_20Hz";
      O     "mainFC3_20Hz";
      );
      =     #mainMustStop;
NETWORK
TITLE =
//запрос останова резервного НА
      O(;
      A     "reserve_started";
      A(;
      O     "second_res_stopped";
      O(;
      L     "PROCESS_DATA".autoCount;
      L     2;
      ==I;
      );
      );
      A(;
      O(;
      A(;
      L     "PROCESS_DATA".offHz2nd;
      L     "FCs".fc1_currFreq;
      >R;
      );
      A(;
      L     "PROCESS_DATA".offHz2nd;
      L     "FCs".fc2_currFreq;
      >R;
      );
      A(;
      L     "PROCESS_DATA".offHz2nd;
      L     "FCs".fc3_currFreq;
      >R;
      );
      );
      O     "highPressTimer";
      );
      );
      O(;
      A     #resConOut;
      AN    #resMustStart;
      );
      O     #mainMustStop;
      =     #resMustStop;
NETWORK
TITLE =
//запрос останова второго резервного НА
      O(;
      A     "sReserve_started";
      A(;
      O     "third_res_stopped";
      O(;
      L     "PROCESS_DATA".autoCount;
      L     1;
      ==I;
      );
      );
      A(;
      O(;
      A(;
      L     "PROCESS_DATA".offHz3th;
      L     "FCs".fc1_currFreq;
      >R;
      );
      A(;
      L     "PROCESS_DATA".offHz3th;
      L     "FCs".fc2_currFreq;
      >R;
      );
      A(;
      L     "PROCESS_DATA".offHz3th;
      L     "FCs".fc3_currFreq;
      >R;
      );
      );
      O     "highPressTimer";
      );
      );
      O(;
      A     #sResConOut;
      AN    #sResMustStart;
      );
      O     #resMustStop;
      =     #sResMustStop;
NETWORK
TITLE =
//запрос останова третьего резервного НА
      O(;
      A     #thResStarted;
      A(;
      O(;
      A(;
      L     "PROCESS_DATA".offHz4th;
      L     "FCs".fc1_currFreq;
      >R;
      );
      A(;
      L     "PROCESS_DATA".offHz4th;
      L     "FCs".fc2_currFreq;
      >R;
      );
      A(;
      L     "PROCESS_DATA".offHz4th;
      L     "FCs".fc3_currFreq;
      >R;
      );
      );
      O     "highPressTimer";
      );
      );
      O(;
      A     #thResConOut;
      AN    #thResMustStart;
      );
      O     #sResMustStop;
      =     #thResMustStop;
NETWORK
TITLE =
//запрос запуска основного НА
      O(;
      L     #P_setpoint;
      L     #P_current;
      -R;
      L     1.000000e-01;
      >R;
      );
//O(;
      O(;
      A     #mainConfirm;
      AN    #mainMustStop;
      );
//AN(;
//O #mainFC1_20Hz;
//O #mainFC2_20Hz;		
//O #mainFC3_20Hz;
//);
//);
      =     #mainMustStart;
NETWORK
TITLE =
//запрос запуска резервного НА
      O(;
      A     "lowPressTimer";
      A(;
      O(;
      L     4.800000e+01;
      L     "FCs".fc1_currFreq;
      <R;
      );
      O(;
      L     4.800000e+01;
      L     "FCs".fc2_currFreq;
      <R;
      );
      O(;
      L     4.800000e+01;
      L     "FCs".fc3_currFreq;
      <R;
      );
      );
      A     "main_started";
      );
      O(;
      A     #resConfirm;
      AN    #resMustStop;
      );
      =     #resMustStart;
NETWORK
TITLE =
//запрос запуска второго резервного НА
      O(;
      A     "lowPressTimer";
      A(;
      O(;
      L     4.800000e+01;
      L     "FCs".fc1_currFreq;
      <R;
      );
      O(;
      L     4.800000e+01;
      L     "FCs".fc2_currFreq;
      <R;
      );
      O(;
      L     4.800000e+01;
      L     "FCs".fc3_currFreq;
      <R;
      );
      );
      A     "reserve_started";
      );
      O(;
      A     #sResConfirm;
      AN    #sResMustStop;
      );
      =     #sResMustStart;
NETWORK
TITLE =
//запрос запуска третьего резервного НА
      O(;
      A     "lowPressTimer";
      A(;
      O(;
      L     4.800000e+01;
      L     "FCs".fc1_currFreq;
      <R;
      );
      O(;
      L     4.800000e+01;
      L     "FCs".fc2_currFreq;
      <R;
      );
      O(;
      L     4.800000e+01;
      L     "FCs".fc3_currFreq;
      <R;
      );
      );
      A     "sReserve_started";
      );
      O(;
      A     #thResStarted;
      AN    #thResMustStop;
      );
      =     #thResMustStart;
END_FUNCTION

FUNCTION "FICTION_PRIORITY" : VOID	// FC 302
AUTHOR : rooman
VERSION : 0.1
VAR_INPUT
  p1_iAuto : BOOL ;
  p2_iAuto : BOOL ;
  p3_iAuto : BOOL ;
  p4_iAuto : BOOL ;
  p1_priority : INT ;
  p2_priority : INT ;
  p3_priority : INT ;
  p4_priority : INT ;
  prioScheme1 : BOOL ;	//1-2-3-4
  prioScheme2 : BOOL ;	//3-1-2-4
  prioScheme3 : BOOL ;	//2-3-1-4
  prioScheme4 : BOOL ;	//2-1-3-4
END_VAR
VAR_OUTPUT
  p1_ficPri : INT ;
  p2_ficPri : INT ;
  p3_ficPri : INT ;
  p4_ficPri : INT ;
END_VAR
VAR_TEMP
  p1_tempPrio : INT ;
  p2_tempPrio : INT ;
  p3_tempPrio : INT ;
  p4_tempPrio : INT ;
END_VAR
BEGIN
NETWORK
TITLE =
//копируем текущие приоритеты во временный буффер
      L     #p1_priority;
      T     #p1_tempPrio;
      L     #p2_priority;
      T     #p2_tempPrio;
      L     #p3_priority;
      T     #p3_tempPrio;
      L     #p4_priority;
      T     #p4_tempPrio;
NETWORK
TITLE =  
      A     #prioScheme1;
      JCN   _001;
      A     #p1_iAuto;
      JC    _010;	//если выключен первый НА при схеме один, повышаем приоритеты остальным
      L     5;
      T     #p1_tempPrio;
      L     #p2_tempPrio;
      DEC   1;
      T     #p2_tempPrio;
      L     #p3_tempPrio;
      DEC   1;
      T     #p3_tempPrio;
      L     #p4_tempPrio;
      DEC   1;
      T     #p4_tempPrio;
_010: NOP   0;
      A     #p2_iAuto;
      JC    _011;
      L     5;
      T     #p2_tempPrio;
      L     #p3_tempPrio;
      DEC   1;
      T     #p3_tempPrio;
      L     #p4_tempPrio;
      DEC   1;
      T     #p4_tempPrio;
_011: NOP   0;
      A     #p3_iAuto;
      JC    _012;
      L     5;
      T     #p3_tempPrio;
      L     #p4_tempPrio;
      DEC   1;
      T     #p4_tempPrio;
_012: NOP   0;
      A     #p4_iAuto;
      JC    _013;
      L     5;
      T     #p4_tempPrio;
_013: NOP   0;
_001: NOP   0;
NETWORK
TITLE =
      A     #prioScheme2;
      JCN   _002;
      A     #p2_iAuto;
      JC    _020;
      L     5;
      T     #p2_tempPrio;
      L     #p3_tempPrio;
      DEC   1;
      T     #p3_tempPrio;
      L     #p4_tempPrio;
      DEC   1;
      T     #p4_tempPrio;
      L     #p1_tempPrio;
      DEC   1;
      T     #p1_tempPrio;
_020: NOP   0;
      A     #p3_iAuto;
      JC    _021;
      L     5;
      T     #p3_tempPrio;
      L     #p4_tempPrio;
      DEC   1;
      T     #p4_tempPrio;
      L     #p1_tempPrio;
      DEC   1;
      T     #p1_tempPrio;
_021: NOP   0;
      A     #p1_iAuto;
      JC    _022;
      L     5;
      T     #p1_tempPrio;
      L     #p4_tempPrio;
      DEC   1;
      T     #p4_tempPrio;
_022: NOP   0;
      A     #p4_iAuto;
      JC    _023;
      L     5;
      T     #p4_tempPrio;
_023: NOP   0;
_002: NOP   0;
NETWORK
TITLE =
      A     #prioScheme3;
      JCN   _003;
      A     #p3_iAuto;
      JC    _030;
      L     5;
      T     #p3_tempPrio;
      L     #p4_tempPrio;
      DEC   1;
      T     #p4_tempPrio;
      L     #p1_tempPrio;
      DEC   1;
      T     #p1_tempPrio;
      L     #p2_tempPrio;
      DEC   1;
      T     #p2_tempPrio;
_030: NOP   0;
      A     #p1_iAuto;
      JC    _031;
      L     5;
      T     #p1_tempPrio;
      L     #p4_tempPrio;
      DEC   1;
      T     #p4_tempPrio;
      L     #p2_tempPrio;
      DEC   1;
      T     #p2_tempPrio;
_031: NOP   0;
      A     #p2_iAuto;
      JC    _032;
      L     5;
      T     #p2_tempPrio;
      L     #p4_tempPrio;
      DEC   1;
      T     #p4_tempPrio;
_032: NOP   0;
      A     #p4_iAuto;
      JC    _033;
      L     5;
      T     #p4_tempPrio;
_033: NOP   0;
_003: NOP   0;
NETWORK
TITLE =
      A     #prioScheme4;
      JCN   _004;
      A     #p2_iAuto;	// 28.12.2016		
      JC    _040;
      L     5;
      T     #p2_tempPrio;
      L     #p1_tempPrio;
      DEC   1;
      T     #p1_tempPrio;
      L     #p4_tempPrio;
      DEC   1;
      T     #p4_tempPrio;
      L     #p3_tempPrio;
      DEC   1;
      T     #p3_tempPrio;
_040: NOP   0;
      A     #p1_iAuto;
      JC    _041;
      L     5;
      T     #p1_tempPrio;
      L     #p3_tempPrio;
      DEC   1;
      T     #p3_tempPrio;
      L     #p4_tempPrio;
      DEC   1;
      T     #p4_tempPrio;
_041: NOP   0;
      A     #p3_iAuto;
      JC    _042;
      L     5;
      T     #p3_tempPrio;
      L     #p4_tempPrio;
      DEC   1;
      T     #p4_tempPrio;
_042: NOP   0;
      A     #p4_iAuto;
      JC    _043;
      L     5;
      T     #p4_tempPrio;
_043: NOP   0;
_004: NOP   0;
NETWORK
TITLE =  
      L     #p1_tempPrio;
      T     #p1_ficPri;
      L     #p2_tempPrio;
      T     #p2_ficPri;
      L     #p3_tempPrio;
      T     #p3_ficPri;
      L     #p4_tempPrio;
      T     #p4_ficPri;
END_FUNCTION

FUNCTION "MICROMASTER_4XX" : VOID	// FC 500
//Функция приема/передачи данных преобразователя частоты Микромастер.
//
AUTHOR : CHANt
FAMILY : OTS
NAME : MM_4XX
VERSION : 0.1
VAR_INPUT
  I_Adress : WORD ;	//Адрес частотника для приема данных
  O_Adress : WORD ;	//Адрес частотника для передачи данных
  Num_DB : BLOCK_DB ;	//Номер блока данных
  I_Enable : BOOL ;	//Включить насос
  I_Error_Reset : BOOL ;	//Квитировать аварию
  I_Setpoint : REAL ;	//Уставка частотнику
  I_PE : REAL ;	//Значение датчика давления на выходе коллектора насосной группы
  I_ASU_UPRAVLENIE : BOOL ;	//Управление от контроллера (AG)
  I_CURR_NOM : REAL ;	//Номинальный ток двигателя
  I_PRESS_HLIM : REAL ;	//Верхний  предел датчика давления
END_VAR
VAR_OUTPUT
  O_Freq : REAL ;	//Текущая частота двигателя
  O_Curr : REAL ;	//Текущий ток двигателя
  O_Power_DC : BOOL ;	//Есть напряжение на частотнике
  O_GOTOV_K_VKL : BOOL ;	//Готов к включению
  O_V_RABOTE : BOOL ;	//Работа
  O_ALARM : BOOL ;	//Неисправность активна
  O_BLOK_ACTUAL : BOOL ;	//Блокировка включения активна
  O_WARNING_ACTUAL : BOOL ;	//Предупреждение активно
  O_ASU_WORK : BOOL ;	//Управление AG (PZD-управление)
  O_Rel : BOOL ;	//Есть связь с частотником
END_VAR
VAR_TEMP
  Error_SFC14 : INT ;	//Код ошибки приема
  Error_SFC15 : INT ;	//Код ошибки передачи
  Error_Recive : BOOL ;
  Error_Send : BOOL ;
END_VAR
BEGIN
NETWORK
TITLE =
//Запрос данных от частотника
      OPN   #Num_DB;	//открыть #Num_DB -  текущий блок данных частотника
      CALL  "DPRD_DAT" (
           LADDR                    := #I_Adress,
           RET_VAL                  := #Error_SFC14,
           RECORD                   := P#DBX 0.0 BYTE 8);	//вызвать функцию четния параметров частотника /  загрузить адрес частотника в сети профибас /  результат функции приема данных / записать полученные данные по указателю в текущий блок данных 
      NOP   0;
NETWORK
TITLE =
//Обработка текущей частоты двигателя
      L     DBW 2;	// загрузить значение частоты из слова DBW2
      ITD;	// преобразовать в двойное целое
      DTR;	//преобразовать в плавающую точку
      L     1.638400e+04;	//загрузить диапазон НЕХ=4000 (DEC=16384)
      /R;	//поделить
      L     5.000000e+01;	// загрузить значение шкалы 50 Гц
      *R;	//перемножить
      T     #O_Freq;	//записать в выход функции  #O_Freq 
NETWORK
TITLE =
//Обработка текущего тока двигателя
//65536.0
      L     DBW 4;	// загрузить значение тока из слова DBW4
      ITD;	// преобразовать в двойное целое
      DTR;	//преобразовать в плавающую точку
      L     8.192000e+03;	//загрузить диапазон НЕХ=2000 (DEC=8192)
      /R;	//поделить
      L     #I_CURR_NOM;	// загрузить значение шкалы  из входа  #I_CURR_NOM  
      *R;	//перемножить
      T     #O_Curr;	//записать в выход функции  #O_Curr    
NETWORK
TITLE =
//Обработка напряжения во внутреннем контуре частотника
//Уточнить при пусковых провалах
      L     DBW 6;	// загрузить значение напряжения во внутреннем контуре частотника из слова DBW6
      L     7000;	// загрузить значение шкалы диапазон НЕХ=7000 (Уточнить при пусковых провалах)
      >I;	//сравнить
      =     #O_Power_DC;	// если значение DBW6 то установить признак наличия напряжения   #O_Power_DC  
NETWORK
TITLE =
//Обработка ошибки связи
      L     #Error_SFC14;	//загрузить возвращаемое значение функции SFC14
      L     0;	//загрузить 0
      ==I;	// если значения равны
      =     #Error_Recive;	//то, установить признак - есть связь с частотником  выход 
NETWORK
TITLE =
//Обработка битов состояния частотника
      A     DBX 1.0;	//если есть
      =     #O_GOTOV_K_VKL;	//то, установить признак "Готов к включению"
      NOP   0;
      A     DBX 1.2;	//если есть
      =     #O_V_RABOTE;	//то, установить признак "Привод в работе"
      NOP   0;
      A     DBX 1.3;	//если есть
      =     #O_ALARM;	//то, установить признак "Неисправность активна"
      NOP   0;
      A     DBX 1.6;	//если есть
      =     #O_BLOK_ACTUAL;	//то, установить признак "Блокировка активна"
      NOP   0;
      A     DBX 1.7;	//если есть
      =     #O_WARNING_ACTUAL;	//то, установить признак "Предупреждение активно"
      NOP   0;
      A     DBX 0.1;	//если есть
      =     #O_ASU_WORK;	//то, установить признак "Работаю от контроллера"
      NOP   0;
NETWORK
TITLE =
//Обработка команд на частотник
      A     #I_Enable;	//если есть  "Пуск частотника"
      =     DBX 9.0;	//то, установить DBX    9.0 
      NOP   0;
      A     #I_Error_Reset;	//если есть  "Квитировать неисправность"
      =     DBX 9.7;	//то, установить DBX 9.7     
      NOP   0;
      A     #I_ASU_UPRAVLENIE;	//если есть  "Управление от контроллера"
      =     DBX 8.2;	//то, установить DBX 8.2 
      =     DBX 9.1;	//установлены биты слова управления для корректной работы ПЧ
      =     DBX 9.2;	//назначение битов есть в соответствующем Data Block
      =     DBX 9.3;
      =     DBX 9.4;
      =     DBX 9.5;
      =     DBX 9.6;
      NOP   0;
NETWORK
TITLE =
//Обработка данных для уставки на частотник
//    RND                               //выделить целое число 
      L     #I_Setpoint;	//загрузить уставку в формате плавающей точки
      L     #I_PRESS_HLIM;	//загрузить верхний предел значения давления датчика
      /R;	//поделить значения
      L     1.638400e+04;	//загрузить диапазон НЕХ=4000 (DEC=16384)
      *R;	//перемножить         
      TRUNC;	//выделить целое число 
      T     DBW 10;	//загрузить в слово DBW10 для передачи в частотник
NETWORK
TITLE =
//Обработка датчика давления насосной группы.
      L     #I_PE;
      L     #I_PRESS_HLIM;
      /R;	//поделить значения
      L     1.638400e+04;	//загрузить диапазон НЕХ=4000 (DEC=16384)
      *R;	//перемножить         
      TRUNC;	//выделить целое число 
      T     DBW 12;	//загрузить в слово DBW12 для передачи в частотник
NETWORK
TITLE =
//Передача данных на частотник
      CALL  "DPWR_DAT" (
           LADDR                    := #O_Adress,
           RECORD                   := P#DBX 8.0 BYTE 8,
           RET_VAL                  := #Error_SFC15);	//вызвать функцию передачи данных в частотник / загрузить адрес передачи / по указателю считать и передать данные на частотник / возвращаемый результат работы функции   SFC15
NETWORK
TITLE =
//Обратка статуса передачи данных на частотник  
//
//
      L     #Error_SFC15;	//загрузить возвращаемое значение функции SFC15
      L     0;	//загрузить 0
      ==I;	// если значения равны
      =     #Error_Send;	//то, установить признак - есть связь с частотником 
NETWORK
TITLE =
      O     #Error_Recive;
      O     #Error_Send;
      =     #O_Rel;	//есть связь с частотником
END_FUNCTION

DATA_BLOCK DB 1
TITLE = Значение каналов AI
VERSION : 1.0
  STRUCT
   CH_0 : WORD ;	//P input
   CH_1 : WORD ;	//P output
  END_STRUCT ;	
BEGIN
END_DATA_BLOCK

DATA_BLOCK DB 2
TITLE = Сигнал с преобразователя (в mA)
VERSION : 1.0
  STRUCT
   SE_1 : REAL ;	//P input
   SE_2 : REAL ;	//P output
  END_STRUCT ;	
BEGIN
END_DATA_BLOCK

DATA_BLOCK "PressDB"	// DB 3
VERSION : 1.0
  STRUCT
   actualPressIN : REAL ;
   bottomPresSensIN : REAL ;
   topPresSensIN : REAL ;
   actualPressOUT : REAL ;
   bottomPresSensOUT : REAL ;
   topPresSensOUT : REAL ;
  END_STRUCT ;	
BEGIN
END_DATA_BLOCK

DATA_BLOCK "FCs"	// DB 4
VERSION : 1.0
  STRUCT
   fc1_currFreq : REAL ;
   fc1_currCurr : REAL ;
   fc1_currPowr : REAL ;
   fc1_voltAru : BOOL ;
   fc1_ready : BOOL ;
   fc1_inWork : BOOL ;
   fc1_alarm : BOOL ;
   fc1_block : BOOL ;
   fc1_warning : BOOL ;
   fc1_asu : BOOL ;
   fc1_connect : BOOL ;
   fc2_currFreq : REAL ;
   fc2_currCurr : REAL ;
   fc2_currPowr : REAL ;
   fc2_voltAru : BOOL ;
   fc2_ready : BOOL ;
   fc2_inWork : BOOL ;
   fc2_alarm : BOOL ;
   fc2_block : BOOL ;
   fc2_warning : BOOL ;
   fc2_asu : BOOL ;
   fc2_connect : BOOL ;
   fc3_currFreq : REAL ;
   fc3_currCurr : REAL ;
   fc3_currPowr : REAL ;
   fc3_voltAru : BOOL ;
   fc3_ready : BOOL ;
   fc3_inWork : BOOL ;
   fc3_alarm : BOOL ;
   fc3_block : BOOL ;
   fc3_warning : BOOL ;
   fc3_asu : BOOL ;
   fc3_connect : BOOL ;
  END_STRUCT ;	
BEGIN
END_DATA_BLOCK

DATA_BLOCK DB 13
TITLE = Гидравлика
VERSION : 1.0
  STRUCT
   SetPoint : BOOL ;
   RealTOD : TIME_OF_DAY ;
   RealD : DATE ;
   ToSetTOD : TIME_OF_DAY ;
   ToSetD : DATE ;
  END_STRUCT ;	
BEGIN
END_DATA_BLOCK

DATA_BLOCK "NOMINAL"	// DB 71
AUTHOR : rooman
VERSION : 0.1
  STRUCT
   fc1_nominal : REAL ;
   fc2_nominal : REAL ;
   fc1_upSen : REAL ;
   fc2_upSen : REAL ;
   fc1_alrReset : BOOL ;
   fc2_alrReset : BOOL ;
   fc3_nominal : REAL ;
   fc3_upSen : REAL ;
   fc3_alrReset : BOOL ;
  END_STRUCT ;	
BEGIN
   fc1_nominal := 1.500000e+01;
   fc2_nominal := 1.500000e+01;
   fc1_upSen := 1.000000e+01;
   fc2_upSen := 1.000000e+01;
   fc3_nominal := 1.500000e+01;
   fc3_upSen := 1.000000e+01;
END_DATA_BLOCK

DATA_BLOCK "EtoDBfunc"	// DB 97
TITLE = sovcim
VERSION : 1.0
  STRUCT
   CurPos : INT ;
   PanPos : INT ;
   Allow : BOOL ;
  END_STRUCT ;	
BEGIN
END_DATA_BLOCK

DATA_BLOCK "AtoDBfunc"	// DB 98
TITLE = nemnoshk))0
VERSION : 1.0
  STRUCT
   CurPos : INT ;
   PanPos : INT ;
   Allow : BOOL ;
   Qwit : BOOL ;
  END_STRUCT ;	
BEGIN
END_DATA_BLOCK

DATA_BLOCK "AlarmState"	// DB 99
TITLE = state of stantion's faults
VERSION : 1.0
  STRUCT
   BreakIN : BOOL ;	//1
   ShortIN : BOOL ;	//2
   BreakOUT : BOOL ;	//3
   ShortOUT : BOOL ;	//4
   Fire : BOOL ;	//5
   Security : BOOL ;	//6
   Flood : BOOL ;	//7
   Phase : BOOL ;	//8
   AVR1 : BOOL ;	//9
   AVR2 : BOOL ;	//10
   Mushroom : BOOL ;	//11
   Dryhod : BOOL ;	//12
   Mokryhod : BOOL ;	//13
   fc1_alarm : BOOL ;	//14
   fc2_alarm : BOOL ;	//15
   non1 : BOOL ;	//16
   Pmp1_fault : BOOL ;	//1
   Pmp2_fault : BOOL ;	//2
   non2 : BOOL ;	//3
   non3 : BOOL ;	//4
   non4 : BOOL ;	//5
   non5 : BOOL ;	//6
   non6 : BOOL ;	//7
   non7 : BOOL ;	//8
   non8 : BOOL ;	//9
   non9 : BOOL ;	//10
   non10 : BOOL ;	//11
   non11 : BOOL ;	//12
   non12 : BOOL ;	//13
   non13 : BOOL ;	//14
   non14 : BOOL ;	//15
   non15 : BOOL ;	//16
  END_STRUCT ;	
BEGIN
END_DATA_BLOCK

DATA_BLOCK DB 100
VERSION : 0.1
  STRUCT
   Num_1 : INT ;
   Date_1 : DATE ;
   Time_1 : TIME_OF_DAY ;
   AlarmType_1 : INT ;
   SavLev_1 : REAL ;
   SavCur_1 : REAL ;
   Num_2 : INT ;
   Date_2 : DATE ;
   Time_2 : TIME_OF_DAY ;
   AlarmType_2 : INT ;
   SavLev_2 : REAL ;
   SavCur_2 : REAL ;
   Num_3 : INT ;
   Date_3 : DATE ;
   Time_3 : TIME_OF_DAY ;
   AlarmType_3 : INT ;
   SavLev_3 : REAL ;
   SavCur_3 : REAL ;
   Num_4 : INT ;
   Date_4 : DATE ;
   Time_4 : TIME_OF_DAY ;
   AlarmType_4 : INT ;
   SavLev_4 : REAL ;
   SavCur_4 : REAL ;
   mada1 : BOOL ;
   mada2 : BOOL ;
   mada3 : BOOL ;
   mada4 : BOOL ;
  END_STRUCT ;	
BEGIN
END_DATA_BLOCK

DATA_BLOCK "Alarms"	// DB 101
VERSION : 0.0
  STRUCT
   alrm : ARRAY  [0 .. 100 ] OF STRUCT
    Num : INT ;
    ArDate : DATE ;
    ArTime : TIME_OF_DAY ;
    AlarmType : INT ;
    SavLev : REAL ;
    SavCur : REAL ;
   END_STRUCT ;
  END_STRUCT ;	
BEGIN
END_DATA_BLOCK

DATA_BLOCK "mada"	// DB 102
VERSION : 0.0
  STRUCT
   alrm : ARRAY  [0 .. 100 ] OF BOOL ;
  END_STRUCT ;	
BEGIN
END_DATA_BLOCK

DATA_BLOCK "Events"	// DB 111
VERSION : 0.0
  STRUCT
   alrm : ARRAY  [0 .. 100 ] OF STRUCT
    Num : INT ;
    ArDate : DATE ;
    ArTime : TIME_OF_DAY ;
    AlarmType : INT ;
   END_STRUCT ;
  END_STRUCT ;	
BEGIN
END_DATA_BLOCK

DATA_BLOCK DB 112
VERSION : 0.1
  STRUCT
   Num_1 : INT ;
   Date_1 : DATE ;
   Time_1 : TIME_OF_DAY ;
   EventType_1 : INT ;
   Num_2 : INT ;
   Date_2 : DATE ;
   Time_2 : TIME_OF_DAY ;
   EventType_2 : INT ;
   Num_3 : INT ;
   Date_3 : DATE ;
   Time_3 : TIME_OF_DAY ;
   EventType_3 : INT ;
   Num_4 : INT ;
   Date_4 : DATE ;
   Time_4 : TIME_OF_DAY ;
   EventType_4 : INT ;
  END_STRUCT ;	
BEGIN
END_DATA_BLOCK

DATA_BLOCK "DB_ROTATION"	// DB 200
AUTHOR : rooman
VERSION : 0.1
  STRUCT
   SUN : BOOL ;
   MON : BOOL ;
   TUE : BOOL ;
   WED : BOOL ;
   THU : BOOL ;
   FRI : BOOL ;
   SAT : BOOL ;
   prioScheme_1 : BOOL ;	//1-2-3-4
   prioScheme_2 : BOOL ;	//3-1-2-4
   prioScheme_3 : BOOL ;	//2-3-1-4
   swiTime : TIME_OF_DAY ;
   silentHill : S5TIME ;
   allow : BOOL ;
   prioScheme_4 : BOOL ;	//2-3-4-1
  END_STRUCT ;	
BEGIN
   prioScheme_1 := TRUE;
   silentHill := S5T#10S;
END_DATA_BLOCK

DATA_BLOCK "PROCESS_DATA"	// DB 300
AUTHOR : rooman
VERSION : 0.1
  STRUCT
   p1_priority : INT ;
   p2_priority : INT ;
   p3_priority : INT ;
   delayLow : S5TIME ;
   delayUp : S5TIME ;
   delayPump : S5TIME ;
   P_setpoint : REAL ;
   P_setLowDiff : REAL ;
   P_setUpDiff : REAL ;
   P_deltaFic : REAL ;
   alloDirFreq : REAL ;
   allowSecRes : BOOL ;
   Alarma : BOOL ;
   TwentyHzOffDelay : S5TIME ;
   lowerHz : REAL ;
   offHz3th : REAL ;
   offHz2nd : REAL ;
   p4_priority : INT ;	//26.09.2016
   p1_ficPrio : INT ;
   p2_ficPrio : INT ;
   p3_ficPrio : INT ;
   p4_ficPrio : INT ;
   offHz4th : REAL ;
   autoCount : INT ;	//28.12.2016
  END_STRUCT ;	
BEGIN
   p1_priority := 1;
   p2_priority := 2;
   p3_priority := 3;
   delayLow := S5T#30S;
   delayUp := S5T#30S;
   delayPump := S5T#30S;
   P_setLowDiff := 3.000000e-01;
   P_setUpDiff := 3.000000e-01;
   P_deltaFic := 5.000000e-01;
   alloDirFreq := 1.500000e+01;
   TwentyHzOffDelay := S5T#30S;
   lowerHz := 1.600000e+01;
   offHz3th := 3.000000e+01;
   offHz2nd := 4.000000e+01;
   p4_priority := 4;
   p1_ficPrio := 1;
   p2_ficPrio := 2;
   p3_ficPrio := 3;
   p4_ficPrio := 4;
   offHz4th := 3.000000e+01;
END_DATA_BLOCK

DATA_BLOCK "kagiri"	// DB 302
VERSION : 1.0
  STRUCT
   shitaKagiriNyuu : REAL ;
   ueKagiriShutsu : REAL ;
   suhoyTime : S5TIME ;
  END_STRUCT ;	
BEGIN
   shitaKagiriNyuu := 1.500000e+00;
   ueKagiriShutsu := 9.000000e+00;
   suhoyTime := S5T#10S;
END_DATA_BLOCK

DATA_BLOCK "DB_PUMPOFF"	// DB 303
AUTHOR : rooman
VERSION : 0.1
  STRUCT
   Pmp1off : BOOL ;
   Pmp2off : BOOL ;
   Pmp3off : BOOL ;
   Delay : S5TIME ;
   resetFcAlarm : BOOL ;
   sf_delay : S5TIME ;
   Pmp4off : BOOL ;	//27.09.16
  END_STRUCT ;	
BEGIN
   Delay := S5T#10S;
   sf_delay := S5T#5M;
END_DATA_BLOCK

DATA_BLOCK "MM430_NS1"	// DB 500
AUTHOR : CHANt
FAMILY : OTS
NAME : NS1_MM43
VERSION : 0.1
  STRUCT
   DEVIATION_SETPOINT : BOOL ;	//Бит 08 Рассогласование уставки и фактического значения 0 ДА Deviation setpoint
   ASU_WORK : BOOL ;	//Бит 09 Управление AG (PZD-управление) 1 ДА PZD control 0 NO 1 YES
   MAX_FREQUENCY : BOOL ;	//Бит 10 Достигнута максимальная частота 1 ДА Maximum frequency reached 0 NO 1 YE
   MAX_CURRRNT : BOOL ;	//Бит 11 Предупреждение: граничное значение тока двигателя 0 ДА Warning: Motor cu
   TORMOZ_ACTUAL : BOOL ;	//Бит 12 Тормоз двигателя активен 1 ДА Motor holding brake active 0 NO 1 YES
   OVERLOAD_PRIVOD : BOOL ;	//Бит 13 Перегрузка двигателя 0 ДА Motor overload 0 YES 1 NO
   PRIVOD_RIGHT : BOOL ;	//Бит 14 Правое вращение 1 ДА Motor runs right 0 NO 1 YES
   OVERLOAD_INVERTER : BOOL ;	//Бит 15 Перегрузка вентильного преобразователя частоты 0 ДА Inverter overload 0
   GOTOV_K_VKL : BOOL ;	//Бит 00 Готов к включению 1 ДА Drive ready 0 NO 1 YES
   GOTOV_K_RABOTE : BOOL ;	//Бит 01 Готов к работе 1 ДА Drive ready to run 0 NO 1 YES
   PRIVOD_V_RABOTE : BOOL ;	//Бит 02 Работа/деблокирование импульсов 1 ДА Drive running 0 NO 1 YES
   ALARM_ACTUAL : BOOL ;	//Бит 03 Неисправность активна 1 ДА Drive fault active 0 NO 1 YES
   STOP2_PRIVOD : BOOL ;	//Бит 04 ВЫКЛ2 активно 0 ДА OFF2 active 0 YES 1 NO
   STOP3_PRIVOD : BOOL ;	//Бит 05 ВЫКЛ3 активно 0 ДА OFF3 active 0 YES 1 NO
   BLOK_ACTUAL : BOOL ;	//Бит 06 Блокировка включения активна 1 ДА ON inhibit active 0 NO 1 YES
   WARNING_ACTUAL : BOOL ;	//Бит 07 Предупреждение активно 1 ДА Drive warning active 0 NO 1 YES
   FREQUENCY : WORD ;	//Текущая частота двигателя
   CURRENT : WORD ;	//Текущий ток двигателя
   VOLTAGE_DC : WORD ;	//DC напряжение (если его нет - значит нет входной напруги)
   CLOCKW_INCHING : BOOL ;	//Бит 08 JOG вправо 0 НЕТ 1 ДА
   CCLOCKW_INCHING : BOOL ;	//Бит 09 JOG влево 0 НЕТ 1 ДА
   ASU_UPRAVLENIE : BOOL ;	//Бит 10 Управление от контроллера (AG) 0 НЕТ 1 ДА
   REVERCE : BOOL ;	//Бит 11 Реверсирование 0 НЕТ 1 ДА
   RESERVED : BOOL ;	//Бит 12 RESERVED
   UP_FREQ : BOOL ;	//Бит 13 Потенциометр двигателя вверх 0 НЕТ 1 ДА
   DOWN_FREQ : BOOL ;	//Бит 14 Потенциометр двигателя вниз 0 НЕТ 1 ДА
   LOCAL_REMOTE_CDS : BOOL ;	//Бит 15 CDS Бит (Local/Remote) 0 НЕТ 1 ДА
   PUSK_PRIVOD : BOOL ;	//Бит 00 ВКЛ / ОТКЛ 0 НЕТ 1 ДА
   BREAK2 : BOOL ;	//Бит 01 ОТКЛ2 : Электр. останов. 0 ДА 1 НЕТ
   BREAK3 : BOOL ;	//Бит 02 ОТКЛ3 : Быстрая остановка 0 ДА 1 НЕТ
   DEBLOCK_IMPULSE : BOOL ;	//Бит 03 Деблокировка импульсов 0 НЕТ 1 ДА
   DEBLOCK_RAZGON : BOOL ;	//Бит 04 Деблокировка датчика разгона (HLG) 0 НЕТ 1 ДА
   ENABLE_RFG : BOOL ;	//Бит 05 Запуск HLG 0 НЕТ 1 ДА
   DEBLOCK_SETPOINT : BOOL ;	//Бит 06 Деблокировка заданной величины 0 НЕТ 1 ДА
   KVIT_ALARM : BOOL ;	//Бит 07 Квитирование сбоя 0 НЕТ 1 ДА
   PID_SETPOINT : WORD ;	//Уставка ПИД-регулятору
   RESERVED_3 : WORD ;	//Резервное слово 3
   RESERVED_4 : WORD ;	//Резервное слово 4
  END_STRUCT ;	
BEGIN
END_DATA_BLOCK

DATA_BLOCK DB 501
AUTHOR : CHANt
FAMILY : OTS
NAME : NS1_MM43
VERSION : 0.1
  STRUCT
   DEVIATION_SETPOINT : BOOL ;	//Бит 08 Рассогласование уставки и фактического значения 0 ДА Deviation setpoint
   ASU_WORK : BOOL ;	//Бит 09 Управление AG (PZD-управление) 1 ДА PZD control 0 NO 1 YES
   MAX_FREQUENCY : BOOL ;	//Бит 10 Достигнута максимальная частота 1 ДА Maximum frequency reached 0 NO 1 YE
   MAX_CURRRNT : BOOL ;	//Бит 11 Предупреждение: граничное значение тока двигателя 0 ДА Warning: Motor cu
   TORMOZ_ACTUAL : BOOL ;	//Бит 12 Тормоз двигателя активен 1 ДА Motor holding brake active 0 NO 1 YES
   OVERLOAD_PRIVOD : BOOL ;	//Бит 13 Перегрузка двигателя 0 ДА Motor overload 0 YES 1 NO
   PRIVOD_RIGHT : BOOL ;	//Бит 14 Правое вращение 1 ДА Motor runs right 0 NO 1 YES
   OVERLOAD_INVERTER : BOOL ;	//Бит 15 Перегрузка вентильного преобразователя частоты 0 ДА Inverter overload 0
   GOTOV_K_VKL : BOOL ;	//Бит 00 Готов к включению 1 ДА Drive ready 0 NO 1 YES
   GOTOV_K_RABOTE : BOOL ;	//Бит 01 Готов к работе 1 ДА Drive ready to run 0 NO 1 YES
   PRIVOD_V_RABOTE : BOOL ;	//Бит 02 Работа/деблокирование импульсов 1 ДА Drive running 0 NO 1 YES
   ALARM_ACTUAL : BOOL ;	//Бит 03 Неисправность активна 1 ДА Drive fault active 0 NO 1 YES
   STOP2_PRIVOD : BOOL ;	//Бит 04 ВЫКЛ2 активно 0 ДА OFF2 active 0 YES 1 NO
   STOP3_PRIVOD : BOOL ;	//Бит 05 ВЫКЛ3 активно 0 ДА OFF3 active 0 YES 1 NO
   BLOK_ACTUAL : BOOL ;	//Бит 06 Блокировка включения активна 1 ДА ON inhibit active 0 NO 1 YES
   WARNING_ACTUAL : BOOL ;	//Бит 07 Предупреждение активно 1 ДА Drive warning active 0 NO 1 YES
   FREQUENCY : WORD ;	//Текущая частота двигателя
   CURRENT : WORD ;	//Текущий ток двигателя
   VOLTAGE_DC : WORD ;	//DC напряжение (если его нет - значит нет входной напруги)
   CLOCKW_INCHING : BOOL ;	//Бит 08 JOG вправо 0 НЕТ 1 ДА
   CCLOCKW_INCHING : BOOL ;	//Бит 09 JOG влево 0 НЕТ 1 ДА
   ASU_UPRAVLENIE : BOOL ;	//Бит 10 Управление от контроллера (AG) 0 НЕТ 1 ДА
   REVERCE : BOOL ;	//Бит 11 Реверсирование 0 НЕТ 1 ДА
   RESERVED : BOOL ;	//Бит 12 RESERVED
   UP_FREQ : BOOL ;	//Бит 13 Потенциометр двигателя вверх 0 НЕТ 1 ДА
   DOWN_FREQ : BOOL ;	//Бит 14 Потенциометр двигателя вниз 0 НЕТ 1 ДА
   LOCAL_REMOTE_CDS : BOOL ;	//Бит 15 CDS Бит (Local/Remote) 0 НЕТ 1 ДА
   PUSK_PRIVOD : BOOL ;	//Бит 00 ВКЛ / ОТКЛ 0 НЕТ 1 ДА
   BREAK2 : BOOL ;	//Бит 01 ОТКЛ2 : Электр. останов. 0 ДА 1 НЕТ
   BREAK3 : BOOL ;	//Бит 02 ОТКЛ3 : Быстрая остановка 0 ДА 1 НЕТ
   DEBLOCK_IMPULSE : BOOL ;	//Бит 03 Деблокировка импульсов 0 НЕТ 1 ДА
   DEBLOCK_RAZGON : BOOL ;	//Бит 04 Деблокировка датчика разгона (HLG) 0 НЕТ 1 ДА
   ENABLE_RFG : BOOL ;	//Бит 05 Запуск HLG 0 НЕТ 1 ДА
   DEBLOCK_SETPOINT : BOOL ;	//Бит 06 Деблокировка заданной величины 0 НЕТ 1 ДА
   KVIT_ALARM : BOOL ;	//Бит 07 Квитирование сбоя 0 НЕТ 1 ДА
   PID_SETPOINT : WORD ;	//Уставка ПИД-регулятору
   RESERVED_3 : WORD ;	//Резервное слово 3
   RESERVED_4 : WORD ;	//Резервное слово 4
  END_STRUCT ;	
BEGIN
END_DATA_BLOCK

ORGANIZATION_BLOCK OB 1
TITLE = "Main Program Sweep (Cycle)"
VERSION : 0.1
VAR_TEMP
  OB1_EV_CLASS : BYTE ;	//Bits 0-3 = 1 (Coming event), Bits 4-7 = 1 (Event class 1)
  OB1_SCAN_1 : BYTE ;	//1 (Cold restart scan 1 of OB 1), 3 (Scan 2-n of OB 1)
  OB1_PRIORITY : BYTE ;	//Priority of OB Execution
  OB1_OB_NUMBR : BYTE ;	//1 (Organization block 1, OB1)
  OB1_RESERVED_1 : BYTE ;	//Reserved for system
  OB1_RESERVED_2 : BYTE ;	//Reserved for system
  OB1_PREV_CYCLE : INT ;	//Cycle time of previous OB1 scan (milliseconds)
  OB1_MIN_CYCLE : INT ;	//Minimum cycle time of OB1 (milliseconds)
  OB1_MAX_CYCLE : INT ;	//Maximum cycle time of OB1 (milliseconds)
  OB1_DATE_TIME : DATE_AND_TIME ;	//Date and time OB1 started
  ErrorSFC : INT ;
  pmp2wfcgo : BOOL ;
  pmp3wfcgo : BOOL ;
  Pmp1on : BOOL ;
  Pmp2on : BOOL ;
  Pmp3on : BOOL ;
  Pmp4on : BOOL ;
END_VAR
BEGIN
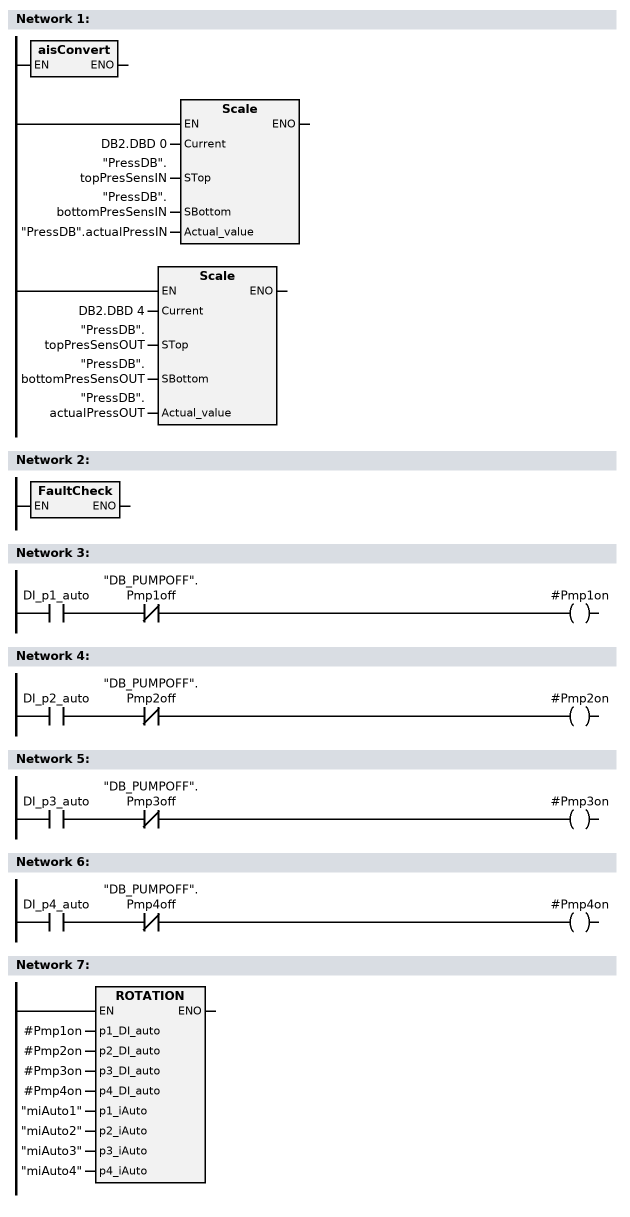
NETWORK
TITLE =
//Обработка аналоговых входов
      CALL  "aisConvert";
      CALL  "Scale" (
           Current                  := DB2.DBD 0,
           STop                     := "PressDB".topPresSensIN,
           SBottom                  := "PressDB".bottomPresSensIN,
           Actual_value             := "PressDB".actualPressIN);
      CALL  "Scale" (
           Current                  := DB2.DBD 4,
           STop                     := "PressDB".topPresSensOUT,
           SBottom                  := "PressDB".bottomPresSensOUT,
           Actual_value             := "PressDB".actualPressOUT);
NETWORK
TITLE =
      CALL  "FaultCheck";
NETWORK
TITLE =
      A     "DI_p1_auto";
      AN    "DB_PUMPOFF".Pmp1off;
      =     #Pmp1on;
NETWORK
TITLE =
      A     "DI_p2_auto";
      AN    "DB_PUMPOFF".Pmp2off;
      =     #Pmp2on;
NETWORK
TITLE =
      A     "DI_p3_auto";
      AN    "DB_PUMPOFF".Pmp3off;
      =     #Pmp3on;
NETWORK
TITLE =
      A     "DI_p4_auto";
      AN    "DB_PUMPOFF".Pmp4off;
      =     #Pmp4on;
NETWORK
TITLE =
      CALL  "ROTATION" (
           p1_DI_auto               := #Pmp1on,
           p2_DI_auto               := #Pmp2on,
           p3_DI_auto               := #Pmp3on,
           p4_DI_auto               := #Pmp4on,
           p1_iAuto                 := "miAuto1",
           p2_iAuto                 := "miAuto2",
           p3_iAuto                 := "miAuto3",
           p4_iAuto                 := "miAuto4");
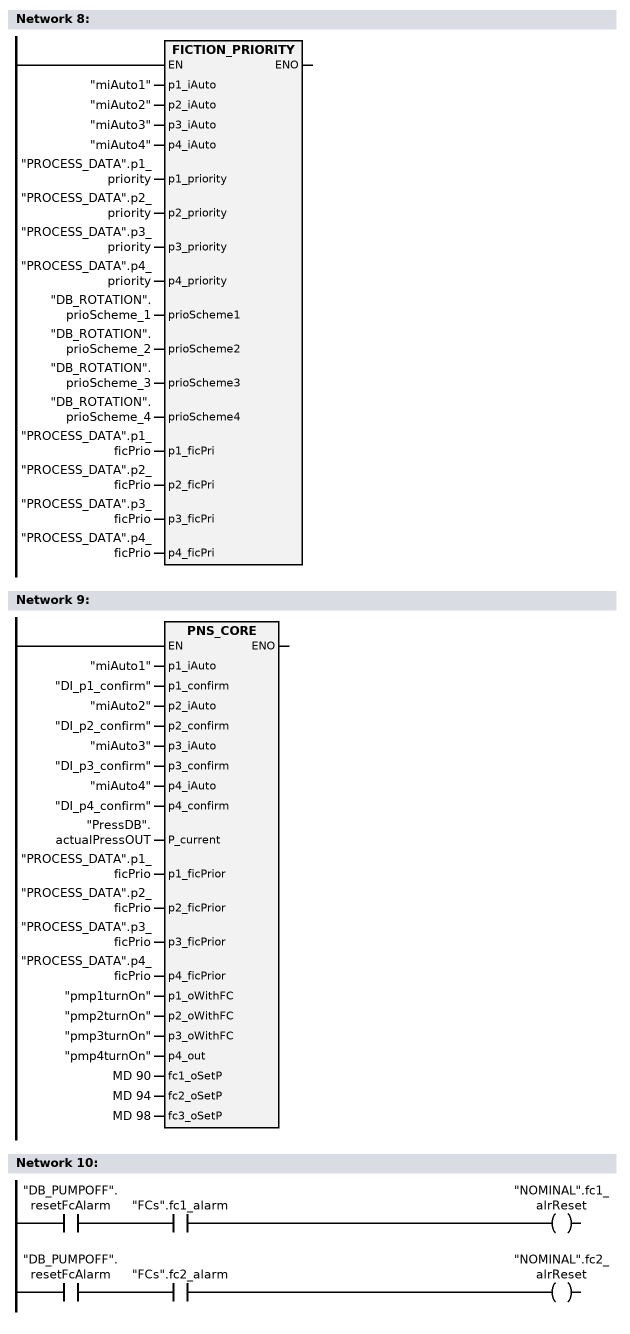
NETWORK
TITLE =
      CALL  "FICTION_PRIORITY" (
           p1_iAuto                 := "miAuto1",
           p2_iAuto                 := "miAuto2",
           p3_iAuto                 := "miAuto3",
           p4_iAuto                 := "miAuto4",
           p1_priority              := "PROCESS_DATA".p1_priority,
           p2_priority              := "PROCESS_DATA".p2_priority,
           p3_priority              := "PROCESS_DATA".p3_priority,
           p4_priority              := "PROCESS_DATA".p4_priority,
           prioScheme1              := "DB_ROTATION".prioScheme_1,
           prioScheme2              := "DB_ROTATION".prioScheme_2,
           prioScheme3              := "DB_ROTATION".prioScheme_3,
           prioScheme4              := "DB_ROTATION".prioScheme_4,
           p1_ficPri                := "PROCESS_DATA".p1_ficPrio,
           p2_ficPri                := "PROCESS_DATA".p2_ficPrio,
           p3_ficPri                := "PROCESS_DATA".p3_ficPrio,
           p4_ficPri                := "PROCESS_DATA".p4_ficPrio);
NETWORK
TITLE =
//CORE
//
      CALL  "PNS_CORE" (
           p1_iAuto                 := "miAuto1",
           p1_confirm               := "DI_p1_confirm",
           p2_iAuto                 := "miAuto2",
           p2_confirm               := "DI_p2_confirm",
           p3_iAuto                 := "miAuto3",
           p3_confirm               := "DI_p3_confirm",
           p4_iAuto                 := "miAuto4",
           p4_confirm               := "DI_p4_confirm",
           P_current                := "PressDB".actualPressOUT,
           p1_ficPrior              := "PROCESS_DATA".p1_ficPrio,
           p2_ficPrior              := "PROCESS_DATA".p2_ficPrio,
           p3_ficPrior              := "PROCESS_DATA".p3_ficPrio,
           p4_ficPrior              := "PROCESS_DATA".p4_ficPrio,
           p1_oWithFC               := "pmp1turnOn",
           p2_oWithFC               := "pmp2turnOn",
           p3_oWithFC               := "pmp3turnOn",
           p4_out                   := "pmp4turnOn",
           fc1_oSetP                := MD 90,
           fc2_oSetP                := MD 94,
           fc3_oSetP                := MD 98);
//       P_current  :="PressDB".actualPressOUT
//       fc1_curFreq:="FCs".fc1_currFreq
//       fc2_curFreq:="FCs".fc2_currFreq
//       p1_oWithFC :="pmp1"
//       p2_oWithFC :="pmp2f"
//       p2_oDirect :="pmp2d"
//       p3_oWithFC :="pmp3f"
//       p3_oDirect :="pmp3d"
//       fc1_oSetP  :=MD90
//       fc2_oSetP  :=MD94
NETWORK
TITLE =
      A     "DB_PUMPOFF".resetFcAlarm;
      A     "FCs".fc1_alarm;
      =     "NOMINAL".fc1_alrReset;
      A     "DB_PUMPOFF".resetFcAlarm;
      A     "FCs".fc2_alarm;
      =     "NOMINAL".fc2_alrReset;
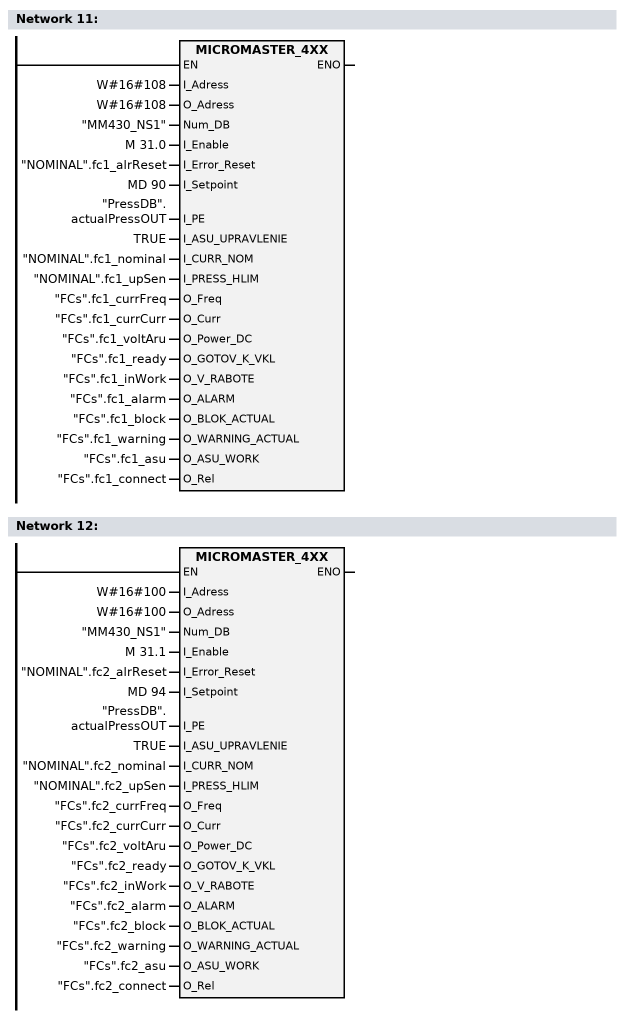
NETWORK
TITLE =
      CALL  "MICROMASTER_4XX" (
           I_Adress                 := W#16#108,
           O_Adress                 := W#16#108,
           Num_DB                   := "MM430_NS1",
           I_Enable                 := M 31.0,
           I_Error_Reset            := "NOMINAL".fc1_alrReset,
           I_Setpoint               := MD 90,
           I_PE                     := "PressDB".actualPressOUT,
           I_ASU_UPRAVLENIE         := TRUE,
           I_CURR_NOM               := "NOMINAL".fc1_nominal,
           I_PRESS_HLIM             := "NOMINAL".fc1_upSen,
           O_Freq                   := "FCs".fc1_currFreq,
           O_Curr                   := "FCs".fc1_currCurr,
           O_Power_DC               := "FCs".fc1_voltAru,
           O_GOTOV_K_VKL            := "FCs".fc1_ready,
           O_V_RABOTE               := "FCs".fc1_inWork,
           O_ALARM                  := "FCs".fc1_alarm,
           O_BLOK_ACTUAL            := "FCs".fc1_block,
           O_WARNING_ACTUAL         := "FCs".fc1_warning,
           O_ASU_WORK               := "FCs".fc1_asu,
           O_Rel                    := "FCs".fc1_connect);
NETWORK
TITLE =
      CALL  "MICROMASTER_4XX" (
           I_Adress                 := W#16#100,
           O_Adress                 := W#16#100,
           Num_DB                   := "MM430_NS1",
           I_Enable                 := M 31.1,
           I_Error_Reset            := "NOMINAL".fc2_alrReset,
           I_Setpoint               := MD 94,
           I_PE                     := "PressDB".actualPressOUT,
           I_ASU_UPRAVLENIE         := TRUE,
           I_CURR_NOM               := "NOMINAL".fc2_nominal,
           I_PRESS_HLIM             := "NOMINAL".fc2_upSen,
           O_Freq                   := "FCs".fc2_currFreq,
           O_Curr                   := "FCs".fc2_currCurr,
           O_Power_DC               := "FCs".fc2_voltAru,
           O_GOTOV_K_VKL            := "FCs".fc2_ready,
           O_V_RABOTE               := "FCs".fc2_inWork,
           O_ALARM                  := "FCs".fc2_alarm,
           O_BLOK_ACTUAL            := "FCs".fc2_block,
           O_WARNING_ACTUAL         := "FCs".fc2_warning,
           O_ASU_WORK               := "FCs".fc2_asu,
           O_Rel                    := "FCs".fc2_connect);
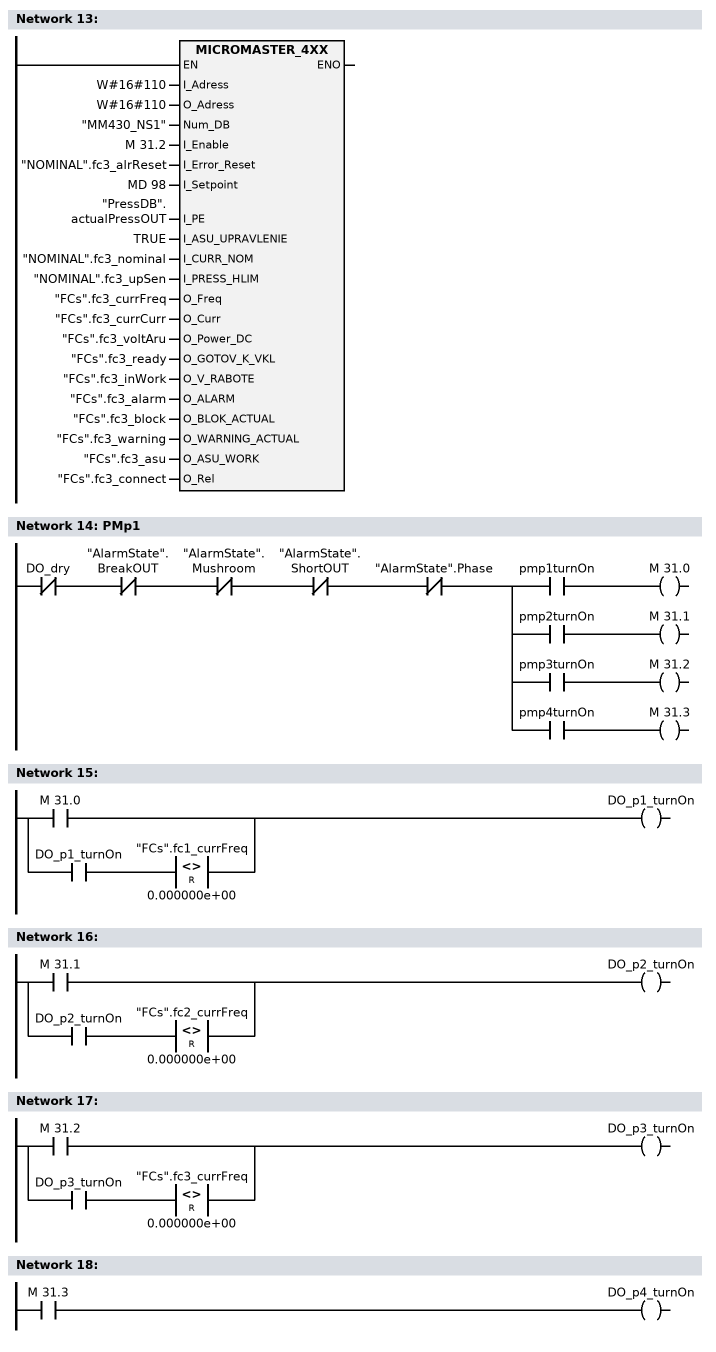
NETWORK
TITLE =
      CALL  "MICROMASTER_4XX" (
           I_Adress                 := W#16#110,
           O_Adress                 := W#16#110,
           Num_DB                   := "MM430_NS1",
           I_Enable                 := M 31.2,
           I_Error_Reset            := "NOMINAL".fc3_alrReset,
           I_Setpoint               := MD 98,
           I_PE                     := "PressDB".actualPressOUT,
           I_ASU_UPRAVLENIE         := TRUE,
           I_CURR_NOM               := "NOMINAL".fc3_nominal,
           I_PRESS_HLIM             := "NOMINAL".fc3_upSen,
           O_Freq                   := "FCs".fc3_currFreq,
           O_Curr                   := "FCs".fc3_currCurr,
           O_Power_DC               := "FCs".fc3_voltAru,
           O_GOTOV_K_VKL            := "FCs".fc3_ready,
           O_V_RABOTE               := "FCs".fc3_inWork,
           O_ALARM                  := "FCs".fc3_alarm,
           O_BLOK_ACTUAL            := "FCs".fc3_block,
           O_WARNING_ACTUAL         := "FCs".fc3_warning,
           O_ASU_WORK               := "FCs".fc3_asu,
           O_Rel                    := "FCs".fc3_connect);
NETWORK
TITLE = PMp1
//12.07.17 AlarmState.Dryhod заменен на DO_dry
      AN    "DO_dry";
      AN    "AlarmState".BreakOUT;
      AN    "AlarmState".Mushroom;
      AN    "AlarmState".ShortOUT;
      AN    "AlarmState".Phase;
      =     L 23.0;
      A     L 23.0;
      A     "pmp1turnOn";
      =     M 31.0;
      A     L 23.0;
      A     "pmp2turnOn";
      =     M 31.1;
      A     L 23.0;
      A     "pmp3turnOn";
      =     M 31.2;
      A     L 23.0;
      A     "pmp4turnOn";
      =     M 31.3;
NETWORK
TITLE =
      O     M 31.0;
      O;
      A     "DO_p1_turnOn";
      A(;
      L     "FCs".fc1_currFreq;
      L     0.000000e+00;
      <>R;
      );
      =     "DO_p1_turnOn";
NETWORK
TITLE =
      O     M 31.1;
      O;
      A     "DO_p2_turnOn";
      A(;
      L     "FCs".fc2_currFreq;
      L     0.000000e+00;
      <>R;
      );
      =     "DO_p2_turnOn";
NETWORK
TITLE =
      O     M 31.2;
      O;
      A     "DO_p3_turnOn";
      A(;
      L     "FCs".fc3_currFreq;
      L     0.000000e+00;
      <>R;
      );
      =     "DO_p3_turnOn";
NETWORK
TITLE =
      A     M 31.3;
      =     "DO_p4_turnOn";
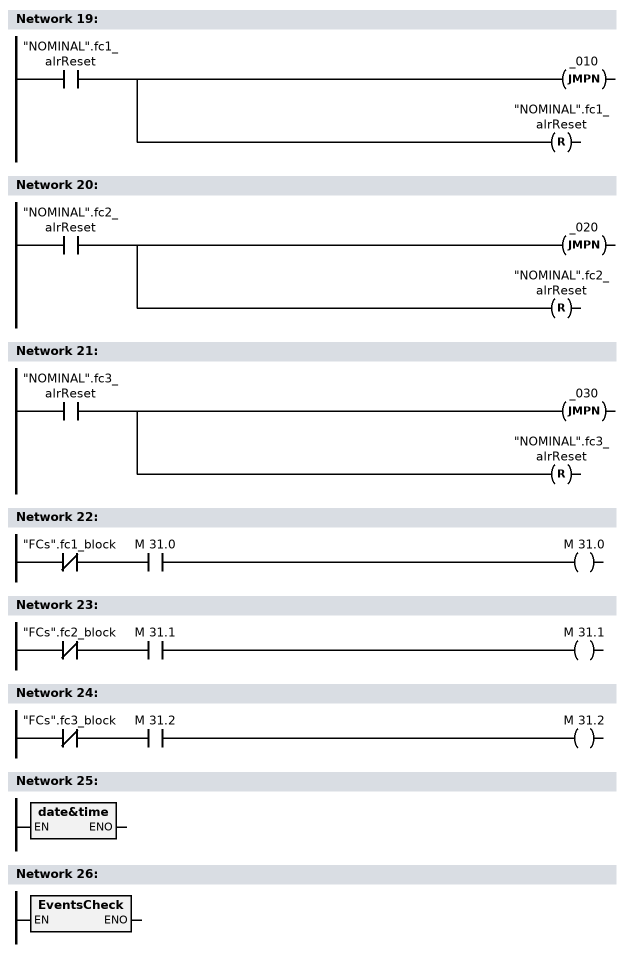
NETWORK
TITLE =
      A     "NOMINAL".fc1_alrReset;
      JCN   _010;
      R     "NOMINAL".fc1_alrReset;
_010: NOP   0;
NETWORK
TITLE =
      A     "NOMINAL".fc2_alrReset;
      JCN   _020;
      R     "NOMINAL".fc2_alrReset;
_020: NOP   0;
NETWORK
TITLE =
      A     "NOMINAL".fc3_alrReset;
      JCN   _030;
      R     "NOMINAL".fc3_alrReset;
_030: NOP   0;
NETWORK
TITLE =
//Reset block FC1
//
      AN    "FCs".fc1_block;
      A     M 31.0;
      =     M 31.0;
NETWORK
TITLE =
//Reset block FC2
//
      AN    "FCs".fc2_block;
      A     M 31.1;
      =     M 31.1;
NETWORK
TITLE =
//Reset block FC2
//
      AN    "FCs".fc3_block;
      A     M 31.2;
      =     M 31.2;
NETWORK
TITLE =
      CALL  "date&time";
NETWORK
TITLE =
      CALL  "EventsCheck";
END_ORGANIZATION_BLOCK
